(* IEC 61131-3 sources: Everest-Indoor-Unit/SWNOVHIDUOUCR00/SWNOVHIDUOUCR00/Sources/Programs, 17 files *)

(* ---- 020_InputMng.st ---- *)
USING System;
USING System.IO;
USING Libs.IOMng_Basic;
USING Libs.Thermodynamic;
(*
    NOTE:
    In order to ADD a new additional function Analog/Digital Input:
        1. INCREASE THE VALUE OF MAXIMUM NUMBER OF IN/OUT CONSTANT DEFINITON (AIN_NO and DIN_NO)
        2. ADD THE NAME AND UOM IN THE RELATIVE UNION STRUCTURE: AinStruct, AinOffsetStruct and DinStruct.
        3. FROM GLOBAL VARIABLE VIEW FLAG THE NEW PROBE AS PARAMETER AND NFC
*)
VAR_GLOBAL CONSTANT
    (* It's not the number of channels available! *)
    (** Max number of possible Analog Inputs *)
    AIN_NO : USINT := 7;
    (* It's not the number of channels available! *)
    (** Max number of possible Digital Inputs *)
    DIN_NO : USINT := 4;
END_VAR

VAR_GLOBAL
    (**Max n° of Ain used by Local board*)
    MAX_AIN_CH  : USINT;
    (**Max n° of Din used by Local board*)
    MAX_DIN_CH  : USINT;
    (**Max n° of Dout used by Local board*)
    MAX_DOUT_CH : USINT;
    (**Max n° of Aout used by Local board*)
    MAX_AOUT_CH : USINT;
    (**Device parameteres (Number of I/O, type o Core...) *)
    HwDesc_1    : HardwareDescription;

    SystemPressure : REAL;
END_VAR

TYPE
    {REGION DIGITAL INPUT CONFIGURATION}
    DinInfoUnion: UNION
        Fct : DinInfoStruct;
        Arr : ARRAY[1..DIN_NO] OF ErrConfig;
    END_UNION;

    DinInfoStruct: STRUCT
        (**Start/Stop Command*)
        RemOnOff        : ErrConfig;
        (**Flow switch*)
        FlowSw          : ErrConfig;
        (**SG input 1*)
        SG1          : ErrConfig;
        (**SG input 2*)
        SG2          : ErrConfig;
    END_STRUCT;

    DinCfgUnion: UNION
        Fct : DinCfgStruct;
        Arr : ARRAY[1..DIN_NO] OF DinConfig;
    END_UNION;

    DinCfgStruct: STRUCT
        (**Start/Stop Command*)
        RemOnOff        : DinConfig;
        (**Flow switch*)
        FlowSw          : DinConfig;
        (**SG input 1*)
        SG1          : DinConfig;
        (**SG input 2*)
        SG2          : DinConfig;
    END_STRUCT;

    DinData: UNION
        Fct : DinStruct;
        Arr : ARRAY[1..DIN_NO] OF BOOL;
    END_UNION;

    DinStruct: STRUCT
        (**Start/Stop Command*)
        RemOnOff        : BOOL;
        (**Flow switch*)
        FlowSw          : BOOL;
        (**SG input 1*)
        SG1          : BOOL := FALSE;
        (**SG input 2*)
        SG2          : BOOL := FALSE;
    END_STRUCT;
    {ENDREGION}

    {REGION ANALOGIC INPUT CONFIGURATION}
    (*
            PAY ATTENTION!!!
            When you add a new AIN remember to also update the MAIN_UI_SEL and AUX_AIN_TYP enumerators.
        *)

    AinInfoUnion: UNION
        Fct : AinInfoStruct;
        Arr : ARRAY[1..AIN_NO] OF ErrConfig;
    END_UNION;

    AinInfoStruct: STRUCT
        (**BT5 DHW bottom temperature*)
        DHWBottomTemp    :   ErrConfig;
        (**BT4 DHW middle temperature*)
        DHWMiddleTemp    :   ErrConfig;
        (**BT3 DHW top temperature*)
        DHWTopTemp       :   ErrConfig;
        (**BT7 DHW supply temperature*)
        DHWSupplyTemp    :   ErrConfig;
        (**BT1 Outdoor temperature*)
        OutDoorTemp    :   ErrConfig;
        (**BT6 Climate system supply temperature*)
        ClimSupplyTemp    :   ErrConfig;
        (**BP1 System pressure*)
        SysPress    :   ErrConfig;
    END_STRUCT;

    AinCfgUnion: UNION
        Fct : AinCfgStruct;
        Arr : ARRAY[1..AIN_NO] OF AinConfig;
    END_UNION;

    AinCfgStruct: STRUCT
        (**BT5 DHW bottom temperature*)
        DHWBottomTemp     :  AinConfig;
        (**BT4 DHW middle temperature*)
        DHWMiddleTemp    :   AinConfig;
        (**BT3 DHW top temperature*)
        DHWTopTemp       :   AinConfig;
        (**BT7 DHW supply temperature*)
        DHWSupplyTemp    :   AinConfig;
        (**BT1 Outdoor temperature*)
        OutDoorTemp    :   AinConfig;
        (**BT7 Climate system supply temperature*)
        ClimSupplyTemp    :   AinConfig;
        (**BP1 System pressure*)
        SysPress    :   AinConfig;
    END_STRUCT;

    AinData: UNION
        Fct : AinDataStruct;
        Arr : ARRAY[1..AIN_NO] OF REAL;
    END_UNION;

    AinDataStruct: STRUCT
        {ATTRIBUTE UOM CELSIUS}
        {METADATA MAX_VAL 999.9}
        {METADATA MIN_VAL -99.9}
        (**BT5 DHW bottom temperature*)
        DHWBottomTemp       :   REAL;
        {ATTRIBUTE UOM CELSIUS}
        {METADATA MAX_VAL 999.9}
        {METADATA MIN_VAL -99.9}
        (**BT4 DHW middle temperature*)
        DHWMiddleTemp      :   REAL;
        {ATTRIBUTE UOM CELSIUS}
        {METADATA MAX_VAL 999.9}
        {METADATA MIN_VAL -99.9}
        (**BT3 DHW top temperature*)
        DHWTopTemp      :   REAL;
        {ATTRIBUTE UOM CELSIUS}
        {METADATA MAX_VAL 999.9}
        {METADATA MIN_VAL -99.9}
        (**BT7 DHW supply temperature*)
        DHWSupplyTemp      :   REAL;
        {ATTRIBUTE UOM CELSIUS}
        {METADATA MAX_VAL 999.9}
        {METADATA MIN_VAL -99.9}
        (**BT1 Outdoor temperature*)
        OutDoorTemp      :   REAL;
        {ATTRIBUTE UOM CELSIUS}
        {METADATA MAX_VAL 999.9}
        {METADATA MIN_VAL -99.9}
        (**BT6 Climate system supply temperature*)
        ClimSupplyTemp    :   REAL;
        {ATTRIBUTE UOM BAR}
        {METADATA MAX_VAL 7.0}
        {METADATA MIN_VAL -1.0}
        (**BP1 System pressure*)
        SysPress    :   REAL;
    END_STRUCT;

    AinOffset: UNION
        Fct : AinOffSetStruct;
        Arr : ARRAY[1..AIN_NO] OF REAL;
    END_UNION;

    AinOffSetStruct: STRUCT
        {ATTRIBUTE UOM DELTACELSIUS}
        (**BT5 DHW bottom temperature*)
        DHWBottomTemp      :   REAL;
        {ATTRIBUTE UOM DELTACELSIUS}
        (**BT4 DHW middle temperature*)
        DHWMiddleTemp      :   REAL;
        {ATTRIBUTE UOM DELTACELSIUS}
        (**BT3 DHW top temperature*)
        DHWTopTemp         :   REAL;
        {ATTRIBUTE UOM DELTACELSIUS}
        (**BT7 DHW supply temperature*)
        DHWSupplyTemp      :   REAL;
        {ATTRIBUTE UOM DELTACELSIUS}
        (**BT1 Outdoor temperature*)
        OutDoorTemp        :   REAL;
        {ATTRIBUTE UOM DELTACELSIUS}
        (**BT6 Climate system supply temperature*)
        ClimSupplyTemp     :   REAL;
        {ATTRIBUTE UOM BAR}
        (**BP1 System pressure*)
        SysPress           :   REAL;
    END_STRUCT;

    {ENDREGION}
END_TYPE

VAR_GLOBAL PERSISTENT
        ReservedIOCfg :BOOL := TRUE;
        Din_Cfg     : DinCfgUnion  := (Fct := (
            (**StartStop*)
            RemOnOff        := (Ch := 0, ModeType := MODE_TYPE_DIN#LIB_IO_DIN),
            (**Flow switch*)
            FlowSw          := (Ch := 0, ModeType := MODE_TYPE_DIN#LIB_IO_DIN),
            (**SG input 1*)
            SG1          := (Ch := 4, ModeType := MODE_TYPE_DIN#LIB_IO_DIN, logic := TRUE),
            (**SG input 2*)
            SG2          := (Ch := 5, ModeType := MODE_TYPE_DIN#LIB_IO_DIN, logic := TRUE)
        ));

        Ain_Cfg     : AinCfgUnion := (Fct := (
            (**DHW bottom temperature*)
            DHWBottomTemp       := (Ch := 5,  ModeType := MODE_TYPE_AIN#LIB_IO_PROBE_NTC),
            (**DHW middle temperature*)
            DHWMiddleTemp       := (Ch := 4,  ModeType := MODE_TYPE_AIN#LIB_IO_PROBE_NTC),
            (**DHW top temperature*)
            DHWTopTemp          := (Ch := 3,  ModeType := MODE_TYPE_AIN#LIB_IO_PROBE_NTC),
            (**DHW supply temperature*)
            DHWSupplyTemp       := (Ch := 6,  ModeType := MODE_TYPE_AIN#LIB_IO_PROBE_NTC),
            (**Outdoor temperature*)
            OutDoorTemp         := (Ch := 1,  ModeType := MODE_TYPE_AIN#LIB_IO_PROBE_NTC),
            (**Climate system supply temperature*)
            ClimSupplyTemp      := (Ch := 2,  ModeType := MODE_TYPE_AIN#LIB_IO_PROBE_NTC),
            (**System pressure*)
            SysPress            := (Ch := 10,  ModeType := MODE_TYPE_AIN#LIB_IO_PROBE_4_20MA)
        ));

    Ain_Min     : AinData := (Fct := (
        SysPress := 0
    ));

    Ain_Max     : AinData := (Fct := (
        SysPress := 6

    ));

    Ain_Offset  : AinOffset :=();

    (**Probe alarm delay*)
    {ATTRIBUTE UOM SECOND}
    PrbAlrm_DT : UINT(0..999) := 10;
END_VAR

PROGRAM InputMng
    VAR_TEMP
        i : DINT;
    END_VAR

    (*All the Programs are skipped while the default valeus are being installed*)
    IF RestoreDefault THEN
        RETURN;
    END_IF;

    {REGION Analog Input Enable}
        Ain_Cfg.Fct.DHWBottomTemp.Enable := TRUE;
        Ain_Cfg.Fct.DHWMiddleTemp.Enable := TRUE;
        Ain_Cfg.Fct.DHWTopTemp.Enable := TRUE;
        Ain_Cfg.Fct.DHWSupplyTemp.Enable := TRUE;
        Ain_Cfg.Fct.ClimSupplyTemp.Enable := TRUE;
        Ain_Cfg.Fct.OutDoorTemp.Enable := TRUE;
        Ain_Cfg.Fct.SysPress.Enable := TRUE;
    {ENDREGION}

    {REGION Digital Input Enable}
        Din_Cfg.Fct.RemOnOff.Enable := TRUE;
        Din_Cfg.Fct.FlowSw.Enable := TRUE;
        Din_Cfg.Fct.SG1.Enable := TRUE;
        Din_Cfg.Fct.SG2.Enable := TRUE;
    {ENDREGION}

    (*Initialization Probe Alarm Delay*)
    FOR i := LOWER_BOUND(Ain_Cfg.Arr, 1) TO UPPER_BOUND(Ain_Cfg.Arr, 1) DO
        Ain_Cfg.Arr[i].AlrmDT := TO_UDINT(PrbAlrm_DT);
    END_FOR;

    IO_Mng.Read(
        BOARD_TYPE#PCO,
        ID,
        U,
        Din_Cfg.Arr,
        Ain_Cfg.Arr,
        Ain_Max.Arr,
        Ain_Min.Arr,
        Ain_Offset.Arr,
        Din_Data.Arr,
        Din_Info.Arr,
        Ain_Data.Arr,
        Ain_Info.Arr,
        uConfig
    );

    HandleSpecialID(1, LIB_IO_PROBE_U_FREQ, 5, uID1);
    WaterFlow_DHW2 := (TO_REAL(uID1.ui) * 0.0106);    // 530 pulses per litre

    HandleSpecialID(2, LIB_IO_PROBE_U_FREQ, 5, uID2);
    WaterFlow_DHW := (TO_REAL(uID2.ui) * 0.0106);    // 530 pulses per litre

    SystemPressure := To_Real(U[10].ud);
    SystemPressure := To_Real(U[10].ui);
    SystemPressure := To_Real(U[10].b);
    SystemPressure := To_Real(U[10].r);
END_PROGRAM

(* ---- 031_StoreAlarms.st ---- *)
USING System;
USING System.Alarm;
USING System.Timer;
USING System.Math;

USING Libs.Logics;
USING Libs.Alarm_Mng;

TYPE
    (**This structure manages all unit's alarms*)
    AlarmUnion : UNION
        (**Array of FBs Alarm_Req*)
        Arr   : ARRAY [1..noAlrms] OF Alarm_Req;
        (**Table of all alarms and them property*)
        Table : AlarmsStruct;
    END_UNION;

    (**List all alarms and them property (Code, Category, Reset type, ...)*)
    AlarmsStruct : STRUCT
        (**Error in number of permanent memory writes*)
        Al_RetainMemNo : Alarm_Req           	 :=	 (StrCode := 'A01', Info := (Code := 001, Category := CAT_AL_SRS_UNIT, Reset := AlarmResetType#Manual));
        (**DHW bottom temperature*)
        Al_DHWBottomTemp : Alarm_Req             :=  (StrCode := 'A02', Info := (Code := 002, Category := CAT_AL_SRS_UNIT, Reset := AlarmResetType#Auto));
        (**DHW middle temperature*)
        Al_DHWMiddleTemp : Alarm_Req             :=  (StrCode := 'A03', Info := (Code := 003, Category := CAT_AL_SRS_UNIT, Reset := AlarmResetType#Auto));
        (**DHW top temperature*)
        Al_DHWTopTemp : Alarm_Req                :=  (StrCode := 'A04', Info := (Code := 004, Category := CAT_AL_SRS_UNIT, Reset := AlarmResetType#Auto));
        (**DHW supply temperature*)
        Al_DHWSupplyTemp : Alarm_Req             :=  (StrCode := 'A05', Info := (Code := 005, Category := CAT_AL_SRS_UNIT, Reset := AlarmResetType#Auto));
        (**Outdoor temperature*)
        Al_OutDoorTemp    :   Alarm_Req          :=  (StrCode := 'A06', Info := (Code := 006, Category := CAT_AL_SRS_UNIT, Reset := AlarmResetType#Auto));
        (**Climate system supply temperature*)
        Al_ClimSupplyTemp    :   Alarm_Req       :=  (StrCode := 'A07', Info := (Code := 007, Category := CAT_AL_SRS_UNIT, Reset := AlarmResetType#Auto));
        (**System pressure*)
        Al_SysPress    :   Alarm_Req             :=  (StrCode := 'A08', Info := (Code := 008, Category := CAT_AL_SRS_UNIT, Reset := AlarmResetType#Auto));
        (**Outdoor unit offline*)
        Al_OUOffline   : Alarm_Req               :=  (StrCode := 'A09', Info := (Code := 009, Category := CAT_AL_SRS_UNIT, Reset := AlarmResetType#Auto));
        (**FreezeProtectionActive*)
        Al_FreezeProAct   : Alarm_Req            :=  (StrCode := 'A10', Info := (Code := 010, Category := CAT_AL_SRS_UNIT, Reset := AlarmResetType#Auto));
    END_STRUCT;
END_TYPE

VAR_GLOBAL CONSTANT
    {REGION UPDATE EVERY TIME AN ALARM IS ADDEDD!}
        (**Number of alarm saved inside ALARM table.
         *NOTE: update every time an alarm is addedd!
        *)
        noAlrms : UINT := 28;
    {ENDREGION}

    {REGION ALARM LOG CONFIGURATION}
        (**Number of logs of alarms saved inside ALARM-LOG table*)
        noAlrmsLog     : UINT := 20;
        (**
         *Size of the array VARs_TO_LOG.
         *Number of additionals variables saved inside ALARM-LOG table,
         *when an alarm is triggered (NOTE: used inside System.Alarm library)
        *)
        MaxAlarmValues : UINT := 0;
    {ENDREGION}

    {REGION CONFIGURE HERE YOUR ALARMs CATEGORY (max 16). YOU NEED TO USE "ActAlr_ForCategory".}
    (**Alarm category associate to ActAlr_ForCategory BIT_0 *) CAT_AL_SRS_UNIT          : UINT := 1;
    (**Alarm category associate to ActAlr_ForCategory BIT_1 *) CAT_AL_SRS_CIRC1         : UINT := 2;
    (**Alarm category associate to ActAlr_ForCategory BIT_2 *) CAT_WARN_CIRC1           : UINT := 4;
    (**Alarm category associate to ActAlr_ForCategory BIT_3 *) SENSOR                   : UINT := 8;
    (**Alarm category associate to ActAlr_ForCategory BIT_4 *) HEATPUMP                 : UINT := 16;
    (**Alarm category associate to ActAlr_ForCategory BIT_5 *) FREE_0                   : UINT := 32;
    (**Alarm category associate to ActAlr_ForCategory BIT_6 *) FREE_1                   : UINT := 64;
    (**Alarm category associate to ActAlr_ForCategory BIT_7 *) FREE_2                   : UINT := 128;
    (**Alarm category associate to ActAlr_ForCategory BIT_8 *) FREE_3                   : UINT := 256;
    (**Alarm category associate to ActAlr_ForCategory BIT_9 *) FREE_4                   : UINT := 512;
    (**Alarm category associate to ActAlr_ForCategory BIT_10*) FREE_5                   : UINT := 1024;
    (**Alarm category associate to ActAlr_ForCategory BIT_11*) FREE_6                   : UINT := 2048;
    (**Alarm category associate to ActAlr_ForCategory BIT_12*) FREE_7                   : UINT := 4096;
    (**Alarm category associate to ActAlr_ForCategory BIT_13*) FREE_8                   : UINT := 8192;
    (**Alarm category associate to ActAlr_ForCategory BIT_14*) FREE_9                   : UINT := 16384;
    (**Alarm category associate to ActAlr_ForCategory BIT_15*) FREE_10                  : UINT := 32768;
    {ENDREGION}
END_VAR

VAR_GLOBAL PERSISTENT
    (**Log alarm array*)
    Log_Alarm  : ARRAY[1..noAlrmsLog] OF AlarmLog;
    (**Index of Log_Alarm *)
    LogAlrmIdx : UINT;
END_VAR

VAR_GLOBAL
    {REGION ALARMS MANAGEMENT}
        (**Container of Alarms table*)
        Alarms              : AlarmUnion;
        (**Array of active alarms*)
        Active_Alrm         : ARRAY[1..noAlrms] OF UINT;
        (**Active alarm status for each category, max 16 differents category (Bit15..Bit0)*)
        ActAlr_ForCategory  : WORD;
    {ENDREGION}

    {REGION ALARMS LOG}
        (**Array of variables to store inside LOG_ALARM array, when an alarm happen*)
        VARs_TO_LOG : ARRAY[0..MaxAlarmValues] OF AlarmValue;
        (**Empty structured used to clean LOG_ALARM array*)
        CleanLog    : AlarmLog;
    {ENDREGION}
END_VAR

VAR_GLOBAL INTERNAL
    (*Used by Modbus files transfer protocol*)
    AlrmInfoArr : ARRAY [1..noAlrms] OF AlarmInfo;
END_VAR

(**This program manages alarm categories and detects the alarms*)
PROGRAM StoreAlarms
    VAR_TEMP
        (**Numeber of alarm active*)
        TotActAlm : UINT;
    END_VAR

    VAR
        (**Array index*)
        idx             : DINT;
        (**Numeber of alarm active in previous cycle*)
        TotActAlm_Old   : UINT;
        TP_ResAlrmByBMS : TP;

        {REGION USED BY LOG-ALARM TO STORE THE "ADDITIONAL VARIABLES"}
        (**A42 trigger used to store additional values*)
        RFtrg_Alr1          : RF_TRIG;
        (**A48 trigger used to store additional values*)
        RFtrg_Alr2          : RF_TRIG;
        (**A46 trigger used to store additional values*)
        RFtrg_Alr3          : RF_TRIG;
        (**A43 trigger used to store additional values*)
        RFtrg_Alr4          : RF_TRIG;
        (**A01 trigger used to store additional values*)
        RFtrg_Alr5          : RF_TRIG;
        (**A35 trigger used to store additional values*)
        RFtrg_Alr6          : RF_TRIG;
        (**A32 trigger used to store additional values*)
        RFtrg_Alr7          : RF_TRIG;
        (**A33 trigger used to store additional values*)
        RFtrg_Alr8          : RF_TRIG;
        (**A37 trigger used to store additional values*)
        RFtrg_Alr9          : RF_TRIG;
        (**A34 trigger used to store additional values*)
        RFtrg_Alr10         : RF_TRIG;
        {ENDREGION}
    END_VAR

    (*Alarm management is be skipped while the default valeus are being installed OR at startup while I/O are being read*)
    IF RestoreDefault OR UnitStatus = UNIT_STATUS#Wait THEN
        RETURN;
    END_IF;

    {REGION RESET ALARM ARRAY}
    TP_ResAlrmByBMS(IN := ResAlrmByBMS, PT := T#5s);        (*Request of reset by BMS*)
    ResAlrmByBMS := TP_ResAlrmByBMS.Q;

    AlrmRes := ResAlrmByBMS OR ResAlrmByHMI;
    {ENDREGION}

    {REGION CLEAN THE LOG ARRAY}
    IF LogAlrmRes THEN
        LogAlrmRes       := FALSE;
        (*RESTART LOG*)
        LogAlrmIdx := 0;

        (*CLEAR LOG LIST*)
        FOR idx := 1 TO TO_DINT(UPPER_BOUND(Log_Alarm, 1)) DO
            Log_Alarm[idx] := CleanLog;
        END_FOR;
    END_IF;
    {ENDREGION}

    {REGION SET DYNAMIQUE CATEGORY}

    {ENDREGION}

    {REGION GET ACTIVE ALARMS}
    FOR idx := 1 TO UPPER_BOUND(Alarms.Arr, 1) DO
        (*Copy the alarm info into a dedicated array*)
        AlrmInfoArr[idx] := Alarms.Arr[idx].Info;

        {REGION "ADDITIONAL VARIABLES" stored inside LOG_ALARM array, when an alarm happen}
		/*IF Alarms.Arr[idx].Info.Code = Alarms.Table.Al_Envelope_Circ1.Info.Code THEN
			RFtrg_Alr1(CLK := Alarms.Arr[idx].Info.Trigger);
            IF RFtrg_Alr1.Q THEN
                VARs_TO_LOG[0].UINT := TO_UINT(0);
            END_IF;*/
		/*ELSIF Alarms.Arr[idx].Info.Code = Alarms.Table.Al_Inv_Circ1.Info.Code THEN
			RFtrg_Alr2(CLK := Alarms.Arr[idx].Info.Trigger);
            IF RFtrg_Alr2.Q THEN
                    VARs_TO_LOG[0].UINT := PWRP_ErrCode_Circ1;
            END_IF;*/
		/*ELSIF Alarms.Arr[idx].Info.Code = Alarms.Table.Al_HiDscgTempComp1_Circ1.Info.Code THEN
        	RFtrg_Alr3(CLK := Alarms.Arr[idx].Info.Trigger);
            IF RFtrg_Alr3.Q THEN
                VARs_TO_LOG[0].UINT := TO_UINT(DscgT_Zone_Circ1);
            END_IF;*/
		/*ELSIF Alarms.Arr[idx].Info.Code = Alarms.Table.Al_DisStartDp_Circ1.Info.Code THEN
			RFtrg_Alr4(CLK := Alarms.Arr[idx].Info.Trigger);
            IF RFtrg_Alr4.Q THEN
                VARs_TO_LOG[0].REAL := DeltaP_Circ1;
            END_IF;*/
		/*ELSIF Alarms.Arr[idx].Info.Code = Alarms.Table.Al_RetainMemNo.Info.Code THEN
			RFtrg_Alr5(CLK := Alarms.Arr[idx].Info.Trigger);
            IF RFtrg_Alr5.Q THEN
                VARs_TO_LOG[0].UDINT := TO_UDINT(RetainMemWrites);
            END_IF;*/
		/*ELSIF Alarms.Arr[idx].Info.Code = Alarms.Table.Al_EEV_Circ1.Info.Code THEN
			RFtrg_Alr6(CLK := Alarms.Arr[idx].Info.Trigger);
            IF RFtrg_Alr6.Q THEN
                VARs_TO_LOG[0].UINT := TO_UINT(EEV_AlrmCode_Circ1);
            END_IF;*/
		/*ELSIF Alarms.Arr[idx].Info.Code = Alarms.Table.Al_WkrHrsComp1_Circ1.Info.Code THEN
			RFtrg_Alr7(CLK := Alarms.Arr[idx].Info.Trigger);
            IF RFtrg_Alr7.Q THEN
                VARs_TO_LOG[0].UINT := TO_UINT(Comp1Circ1_HrsRetain);
            END_IF;*/
		/*ELSIF Alarms.Arr[idx].Info.Code = Alarms.Table.Al_WkrHrsSrc_Circ1.Info.Code THEN
			RFtrg_Alr10(CLK := Alarms.Arr[idx].Info.Trigger);
            IF RFtrg_Alr10.Q THEN
                VARs_TO_LOG[0].UINT := TO_UINT(Source1Circ1_HrsRetain);
            END_IF;*/
		//END_IF;
        {ENDREGION}

        Alarms.Arr[idx]
                        (
                            DataVal         := VARs_TO_LOG, (* Remember to define ALARM_VALUES *)
                            AlrmRes         := AlrmRes,
                            Lst_ActAlrm     := Active_Alrm,
                            Lst_LogAlrm     := Log_Alarm,
                            Lst_LogAlrm_Idx := LogAlrmIdx
                        );
    END_FOR;
    {ENDREGION}

    {REGION GET ALARM CATEGORIES}
    ActAlr_ForCategory := Alarm_Mng(Active_Alrm);
    Al_SrsUnit            := ActAlr_ForCategory.0;  									// BIT n.0  -> CAT_AL_SRS_UNIT
    Al_SrsCirc1           := ActAlr_ForCategory.1 OR Al_SrsUnit;// BIT n.1  -> Al_SRS_CIRC1
    Wrg_Regul             := ActAlr_ForCategory.4;                      				// BIT n.4  -> CAT_WRG_REGUL
    Wrg_Circ1             := ActAlr_ForCategory.5;                      				// BIT n.7  -> CAT_WRG_CIRC1
    Wrg_HrsCounters       := ActAlr_ForCategory.7;                      				// BIT n.10 -> CAT_WRG_HRSCOUNTER
    {ENDREGION}

    {REGION MANAGEMENT OF ALARM RELAY AND GROUPED ALARMS}
    (*Depending on alarm relay configuration, the alarm relay is activated by serious alarms only or by all alarms (including devices maintenance, retain memory,...) *)
    Al_RegulationAlrms :=    Al_SrsUnit
                          OR Al_SrsCirc1
                          OR Wrg_Regul;

    Al_MiscAlrms :=    Wrg_Circ1
                    OR Wrg_HrsCounters;

    RelayAlrm := Al_RegulationAlrms OR Al_MiscAlrms;
    {ENDREGION}

    {REGION COUNT OF TOTAL ALARMs AND WARNINGs ACTIVE}
    FOR idx := 1 TO TO_DINT(UPPER_BOUND(Active_Alrm,1)) DO
        IF Active_Alrm[idx] >= 1 THEN
            TotActAlm := TotActAlm + 1;
        END_IF;
    END_FOR;

    GblAlarm := UINT_TO_BOOL(TotActAlm);

    (*LED-ALARM and BUZZER*)
    IF TotActAlm > TotActAlm_Old THEN
        Req_FixLED_Alarm   := FALSE;    // LED-ALARM on
        Req_BlinkLED_Alarm := TRUE;     // LED-ALARM is blinking
        BuzzerSilenced     := FALSE;    // Buzzer is buzzing
    END_IF;

    TotActAlm_Old := TotActAlm;
    {ENDREGION}
END_PROGRAM

(* ---- 120_OutputMng.st ---- *)
USING System.IO;
USING System;
USING Libs.Math;
USING Libs.IOMng_Basic;

(*
    NOTE:
    In order to ADD a new additional function Analog/Digital Output:
        1. INCREASE THE VALUE OF MAXIMUM NUMBER OF IN/OUT CONSTANT DEFINITON (MAX_DO_NO and MAX_AO_NO)
        2. ADD THE NAME AND UOM IN THE RELATIVE UNION STRUCTURE: AoutStruct and DoutStruct
        3. FROM GLOBAL VARIABLE VIEW FLAG THE NEW PROBE AS PARAMETER AND NFC
*)
VAR_GLOBAL CONSTANT
    (* It's not the number of channels available! *)
    (** Max number of possible Digital Outputs *)
    MAX_DO_NO   : USINT := 7;
    (* It's not the number of channels available! *)
    (** Max number of possible Analog Outputs *)
    MAX_AO_NO   : USINT := 2;
END_VAR

TYPE
    {REGION ANALOGIC OUTPUT CONFIGURATION}
        AoutInfoUnion: UNION
            Fct : AoutInfoStruct;
            Arr : ARRAY[1..MAX_AO_NO] OF ErrConfig;
        END_UNION;

        AoutInfoStruct: STRUCT
            (**Circulation pump 1*)
            CircPump1    :   ErrConfig;
            (**Circulation pump 2*)
            CircPump2    :   ErrConfig;
        END_STRUCT;

        AoutCfgUnion: UNION
            Fct : AoutCfgStruct;
            Arr : ARRAY[1..MAX_AO_NO] OF AoutConfig;
        END_UNION;

        AoutCfgStruct: STRUCT
            (**Circulation pump 1*)
            CircPump1    :   AoutConfig;
            (**Circulation pump 2*)
            CircPump2    :   AoutConfig;
        END_STRUCT;

        AoutData: UNION
            Fct : AoutStruct;
            Arr : ARRAY[1..MAX_AO_NO] OF REAL;
        END_UNION;

        AoutStruct: STRUCT
            (**Circulation pump 1*)
            {ATTRIBUTE UOM PERCENT}
            CircPump1    :   REAL;
            {ATTRIBUTE UOM PERCENT}
            (**Circulation pump 2*)
            CircPump2    :   REAL;
        END_STRUCT;
    {ENDREGION}

    {REGION DIGITAL OUTPUT CONFIGURATION}
        DoutInfoUnion: UNION
            Fct : DoutInfoStruct;
            Arr : ARRAY [1..MAX_DO_NO] OF ErrConfig;
        END_UNION;

        DoutInfoStruct: STRUCT
            (**General alarm *)
            GlbAl          :   ErrConfig;
            (**Shunt valve*)
            ShuntVlvDout          :   ErrConfig;
            (**Immersion heater step 1*)
            ImmheatStep1   : ErrConfig;
            (**Immersion heater step 2*)
            ImmheatStep2   : ErrConfig;
            (**Immersion heater step 3*)
            ShuntVlvOffDout   : ErrConfig;
            (**Reversing valve*)
            RevVlv         : ErrConfig;
            (**Shut off valve*)
            ShutOffVlv     : ErrConfig;
        END_STRUCT;

        DoutCfgUnion: UNION
            Fct : DoutCfgStruct;
            Arr : ARRAY [1..MAX_DO_NO] OF DoutConfig;
        END_UNION;

        DoutCfgStruct: STRUCT
            (**General alarm *)
            GlbAl          :    DoutConfig;
            (**Shunt valve*)
            ShuntVlvDout          :   DoutConfig;
            (**Immersion heater step 1*)
            ImmheatStep1   : DoutConfig;
            (**Immersion heater step 2*)
            ImmheatStep2   : DoutConfig;
            (**Immersion heater step 3*)
            ShuntVlvOffDout   : DoutConfig;
            (**Reversing valve*)
            RevVlv         : DoutConfig;
            (**Shut off valve*)
            ShutOffVlv     : DoutConfig;
        END_STRUCT;

        DoutData: UNION
            Fct : DoutStruct;
            Arr : ARRAY[1..MAX_DO_NO] OF BOOL;
        END_UNION;

        DoutStruct: STRUCT
            (**General alarm *)
            GlbAl               :   BOOL;
            (**Shunt valve*)
            ShuntVlvDout            :   BOOL;
            (**Immersion heater step 1*)
            ImmheatStep1   : BOOL;
            (**Immersion heater step 2*)
            ImmheatStep2   : BOOL;
            (**Immersion heater step 3*)
            ShuntVlvOffDout   : BOOL;
            (**Reversing valve*)
            RevVlv         : BOOL;
            (**Shut off valve*)
            ShutOffVlv     : BOOL;
        END_STRUCT;
    {ENDREGION}

END_TYPE

VAR_GLOBAL PERSISTENT
    Dout_Cfg        : DoutCfgUnion  := (Fct := (
        (**General alarm *)
        GlbAl               := (Ch := 0),
        (**Shunt valve*)
        ShuntVlvDout        := (Ch := 8),
        (**Immersion heater step 1*)
        ImmheatStep1        := (Ch := 4),
        (**Immersion heater step 2*)
        ImmheatStep2        := (Ch := 5),
        (**Immersion heater step 3*)
        ShuntVlvOffDout     := (Ch := 9),
        (**Reversing valve*)
        RevVlv              := (Ch := 1),
        (**Shut off valve*)
        ShutOffVlv          := (Ch := 7)
    ));

    Aout_Cfg        : AoutCfgUnion := (Fct := (
        (**Circulation pump 1*)
        CircPump1      := (Ch := 3,  ModeType := MODE_TYPE_AOUT#LIB_IO_PWM_2_KHZ),
        (**Circulation pump 2*)
        CircPump2      := (Ch := 4,  ModeType := MODE_TYPE_AOUT#LIB_IO_PWM_2_KHZ)

    ));

    Aout_Min : AoutData :=(Fct := (CircPump1 :=0, CircPump2 := 0));
    Aout_Max : AoutData :=(Fct := (CircPump1 :=100, CircPump2 := 100));
END_VAR

PROGRAM OutputMng
    VAR_TEMP
        i : DINT;
    END_VAR
    (*Enabling Analog outputs*)
    {REGION Analog Output Enable}
        Aout_Cfg.Fct.CircPump1.Enable := TRUE;
        Aout_Cfg.Fct.CircPump2.Enable := TRUE;
    {ENDREGION}

    (*Enabling Digital outputs*)
    {REGION Digital Output Enable}
        Dout_Cfg.Fct.GlbAl.Enable := TRUE;
        Dout_Cfg.Fct.ShuntVlvDout.Enable := TRUE;
        Dout_Cfg.Fct.ImmheatStep1.Enable := ImmHeatStage >= 1;
        Dout_Cfg.Fct.ImmheatStep2.Enable := ImmHeatStage >= 2;
        Dout_Cfg.Fct.ShuntVlvOffDout.Enable := TRUE;
        Dout_Cfg.Fct.RevVlv.Enable := TRUE;
        Dout_Cfg.Fct.ShutOffVlv.Enable  := TRUE;
    {ENDREGION}

	{REGION Analog Output value}
    Aout_Data.Fct.CircPump1 := Circ1Act_Req;
    Aout_Data.Fct.CircPump2 := Circ2Act_Req;
	{ENDREGION}

	{REGION Digital Output Value}
	Dout_Data.Fct.GlbAl := GblAlarm;
    Dout_Data.Fct.ShuntVlvDout := ShuntVlv_On;
    Dout_Data.Fct.ImmheatStep1 := ActImmStep_Out.0;
    Dout_Data.Fct.ImmheatStep2 := ActImmStep_Out.1;
    Dout_Data.Fct.ShuntVlvOffDout := ShuntVlv_Off;
    Dout_Data.Fct.RevVlv       := (DHWReq AND OU_CompOn) OR SWValveManA;
    Dout_Data.Fct.ShutOffVlv   := CoolReq OR ShutOffMan;
	{ENDREGION}
    FOR i := 1 TO UPPER_BOUND(Aout_Data.Arr, 1) DO
        Aout_Data.Arr[i] := ScalerLimited(Aout_Data.Arr[i], 0.0, 100.0, Aout_Min.Arr[i], Aout_Max.Arr[i]);
    END_FOR;

    IO_Mng.Write(
        BOARD_TYPE#PCO,
        Dout_Cfg.Arr,
        Dout_Data.Arr,
        Aout_Cfg.Arr,
        Aout_Data.Arr,
        Dout_Info.Arr,
        Aout_Info.Arr,
        NO,
        noConfig,
        Y,
        yConfig,
        uConfig,
        Uout
    );

END_PROGRAM

(* ---- 010_GENERAL_MNG.st ---- *)
USING System;
USING System.NVRAM;
USING System.Timer;
USING System.Serial;
USING System.Globalization;
USING Libs.GetTime;

PROGRAM Main
    VAR
        (**After restoring the memory to default, it waits 6s before restarting the PLC*)
        TON_WaitRestartPlc  : TON;
        (**R_TRIG Restore Default Settings*)
        Rtrg_RestoreDefault  : R_TRIG;
        (**First cycle done used by NVRAM management*)
        FirstCycleDone_NVRAM : BOOL;
        (**Istance of SoftwareSafeUpload manage the system call GetFullDownloadRequest()*)
        SwSafeUpload         : SoftwareSafeUpload;
        i                    : DINT;
    END_VAR

    VAR_TEMP
        NVRAM_BOOL_Tmp : BYTE;
        TmpTimezone : STRING;
    END_VAR

    RetainMemWrites := GetRetainWritingsNumber();

    TaskMainCurrT   := GetTaskStartTimeAdv();
    TaskMainLiveCnt := GetTaskLiveCounter();
    RetainWrN       := TO_UDINT(GetRetainWritingsNumber());
    TaskMainExeT    := TaskMainCurrT - MemTime;
    MemTime         := TaskMainCurrT;

    {REGION RESTORE MEMORY}
    Rtrg_RestoreDefault(CLK := RestoreDefault);
    (*Saving BMS before restoring memory*)
    IF Rtrg_RestoreDefault.Q THEN
        SPV_Addr_SavedRAM := SPV_Addr;
        SPV_Baud_SavedRAM := SPV_Baud;
        SPV_Conf_SavedRAM := SPV_Conf;
    END_IF;

    IF RestoreDefault AND NOT RetainRestored THEN
        RetainRestoreDefault(); (*NOTE: This request will be executed at END of MAIN task.*)
        RetainRestored := TRUE;
    END_IF;

    //------------------------------------------------------------------------------------
    //------------ WARM SOFTWARE RESET----------------------------------------------------
    //------------------------------------------------------------------------------------
    TON_WaitRestartPlc(IN := RetainRestored, PT := T#6s);

    IF TON_WaitRestartPlc.Q THEN
        // Wait 6s because Retain will be write every 5s
        // 0 - WARM start;
        SoftwareReset(0);
    END_IF;
    {ENDREGION}

    {REGION DATE AND TIME}
    GetLocalTime(LocTime);
    Day_Week := DAY_OF_WEEK(LocTime);

    {REGION SET CLOCK TIME BY APPLICA}
    IF AppSetDateTime THEN
        AppSetDateTime := FALSE; //CS: da provare senza il reset
        //Necessary and in this order
        SetTimeZone(AppTimeZone);
        SetTime(AppDateTime); //APPLICA give UTC Times
        TimezoneIdx := FindTimezoneIndex(TimeZonePOSIX, AppTimeZone);
    END_IF;
    {ENDREGION}

    {REGION SET CLOCK TIME BY USER INTERFACE}
    IF SetClock THEN
        SetClock := FALSE;
        //Necessary and in this order
        SetTimeZone(TimeZonePOSIX[TimezoneIdx]);
        SetLocalTime(CONCAT_DT(
		    TO_UINT(YearIn) + 2000,
		    TO_UINT(MonthIn),
		    TO_UINT(DayIn),
		    TO_UINT(HourIn),
		    TO_UINT(MinuteIn),
		    TO_UINT(SecondIn),
		    0
		));
    END_IF;
    {ENDREGION}
    {ENDREGION}

    {REGION RETAIN WRITING SETTINGS}
    (*This FB manage the "retain writing error" as bios specification. *)
    RetainSetErasureWindowSize(ErasureWindowSize);
    RetainSetErasureWindowsNumber(ErasureWindowsNumber);
    RetainSetMaxErasure(MaxErasure);
    {ENDREGION}

    {REGION SYSTEM INFORMATION}
    IF NOT FirstCycleDone THEN
        MemTime        := TaskMainCurrT;
        GetSystemInfo(SysInfo);
        GetHardwareDescription(HardwareInfo);
        GetModel(DeviceType, BoardType, MachineType, HwCode);
        GetProjectInfo(InfoProject);
        GetProductInfo(InfoProduct);
        GUID := SplitPrjGUID(InfoProject.ProjectID);
        SwVersion := (TO_UINT(InfoProject.VersionMajor) * 10000) + (TO_UINT(InfoProject.VersionMinor) * 1000) + TO_UINT(InfoProject.VersionBuild);
		OS_Version := TO_UINT(SysInfo.FirmwareVersion);
		BootVersion := TO_UINT(SysInfo.BootloaderVersion);

        {REGION COMUNICATION IS STOPPED DURING INITIALIZATION OF INTERNAL PROTOCOLs STRUCTUREs.}
        (*BMS*)
        Supervisor.Init(FALSE);
        (*Fieldbus*)
        MBM_Line.Init(FALSE);
        (*Display*)
        Display.Init();
        {ENDREGION}

        {REGION IoT Third Parts Integration: Alarms retrieved via "Modbus File Transfer"}
        (*Following APIs calls are needed*)
        System.Alarm.AlarmInfoManagement(AlrmInfoArr);
        System.Alarm.AlarmLogManagement(LOG_ALARM);
        {ENDREGION}

        {REGION SAVING OF TIMEZONE WHEN RTC SET BY APPs}
		GetTimeZone(TmpTimezone);
        TimezoneIdx := FindTimezoneIndex(TimeZonePOSIX, TmpTimezone);
        {ENDREGION}
        FirstCycleDone := TRUE;
    END_IF;
    {ENDREGION}

    {REGION SYSTEM CONFIGURAITON}
        //System configuration selection
        //None selected
        // 1: Heating system 1 + DHW
        // 2: Heating system 1 + DHW
        // 3: Heating system 1 + Heating system 2 + DHW
        // 4: Heating system 1 + Cooling + DHW
        // 5: Heating system 1 + Heating system 2 + DHW + Cooling

        IF(SystemCfg > 0)THEN
            SystemCfg_AllowDHW := SystemCfg >= 1;
            SystemCfg_AllowHeat := SystemCfg >= 2;
            SystemCfg_AllowImm := SystemCfg >= 1;
            SystemCfg_AllowCool := SystemCfg >=  4;
            SystemCfg_NoCfgSel := FALSE;
        ELSE
            SystemCfg_AllowDHW := FALSE;
            SystemCfg_AllowHeat := FALSE;
            SystemCfg_AllowImm := FALSE;
            SystemCfg_AllowCool := FALSE;
            SystemCfg_NoCfgSel := TRUE;
        END_IF;
    {ENDREGION}

    {REGION PROTOCOLS}

    {REGION BMS/FIELDBUS SERIAL PORTs CONFIGURATION}
    CASE UoMZoneHMI OF
        UOM_ZONE#SI:
            Supervisor.Info.Zone := SI;
            // Server BMS uses only SI to communicate (Client FielBus <-> Server BMS)
            // NOTE: In a net CLIENT+SERVER set NoConverion =0 beetwen: Client FielBus <-> Server BMS to increase pCO speed
            // i.e.: FBnet.Info.Zone=0 and BMSnet.Info.Zone=0
            Display.Info.Zone := SI;
        UOM_ZONE#Imperial:
            Supervisor.Info.Zone := Imperial;
            Display.Info.Zone := Imperial;
    ELSE
        Supervisor.Info.Zone := NONE;
        Display.Info.Zone := NONE;
    END_CASE;

    {REGION CHANGE BMS2 SETTINGS}
    (*Memory after deleting command is immediately ready the next cycles*)
    IF RetainRestored THEN
        // Restore BMS2 settings
        SPV_Addr := SPV_Addr_SavedRAM;
        SPV_Baud := SPV_Baud_SavedRAM;
        SPV_Conf := SPV_Conf_SavedRAM;

        // Force update BMS2 settings
        SPV_ChangeSet := TRUE;
    END_IF;

    IF SPV_ChangeSet THEN
		Supervisor.Info.TimeOut := TO_UDINT(SPV_OfflineTimeout)*1000;
        SetupSerialSettings(Supervisor.SerialSettings, SPV_Baud, SPV_Conf, getServerPort(SPV_Port));
        Supervisor.ChangeIdent(SPV_Addr);
        // Change setting of BMS supervisor port
        Supervisor.ChangeSettings();
        // Set the same settings for BMS port on Default app (NOTE: In case of FW ugrade the device will be reachable with the previous settings)
        SaveIdePortSettings(Supervisor.SerialSettings.Channel, Supervisor.SerialSettings.Speed, Supervisor.SerialSettings.Bits, Supervisor.SerialSettings.Parity, Supervisor.SerialSettings.Stops, SPV_Addr);

        SPV_ChangeSet := FALSE;
    END_IF;

    SPV_Online := Supervisor.Info.Online;
    {ENDREGION}

    {REGION CHANGE FIELDBUS2 SETTINGS}
    IF FB2_ChangeSet THEN
        SetupSerialSettings(MBM_Line.SerialSettings, FB2_Baud, FB2_Conf, getClientPort(MBM_Line_Port));
        // Change setting of FB supervisor port
        MBM_Line.ChangeSettings();

        FB2_ChangeSet := FALSE;
    END_IF;
    {ENDREGION}
    {ENDREGION}

    {REGION READ BUFFER OF EACH SERIAL PORT}
    // NOTE: when the protocols are in START the read() method obtain the variables
    //       from each buffer -> so the variables can be used inside STone.

    // BMS
    Supervisor.Read();
    // Fieldbus
    MBM_Line.Read();
    Display.Read();
	{IF DEF (PGD)}
    	TerminalDetector.Run(Display);
	{ENDIF}
    {ENDREGION}
	{ENDREGION}

    {REGION NVRAM management}
    IF NOT FirstCycleDone_NVRAM THEN

        /*NVRAM_ReadVar(1, NVRAM_BOOL_Tmp);
        Dout_FourWVlv_NVRAM := TO_BOOL(NVRAM_BOOL_Tmp);

        FirstCycleDone_NVRAM := TRUE;
    ELSE
        NVRAM_WriteVar(1, TO_BYTE(Dout_FourWVlv_NVRAM));*/
    END_IF;
    {ENDREGION}

    //Outdoor unit status management
    OU_Online := OU_Unit.Info.isOnline;

    (*Call of SoftwareSafeUpload manage the system call GetFullDownloadRequest()*)
    SwSafeUpload(
        KeybOffOn := BmsOnOff,
        StartUpload := UnitOff
    );
END_PROGRAM

(* ---- 030_AlarmsMng.st ---- *)
USING System;
USING System.Timer;
USING Libs.Timer;

PROGRAM AlarmsMng
	VAR
	    RTrig_RetainErr : R_TRIG;
	END_VAR

    (*Alarm management is skipped while the default valeus are being installed OR at startup while I/O are being read*)
    IF RestoreDefault OR UnitStatus = UNIT_STATUS#Wait THEN
        RETURN;
    END_IF;

	RTrig_RetainErr(
		CLK := ExceptionInstance.ExceptionError = ERR_RETAIN_SAVE_TOO_OFTEN
	);
	Alarms.Table.Al_RetainMemNo.Info.Trigger := RTrig_RetainErr.Q;

    {REGION UNIT ALARMS BY DIN}
    {ENDREGION}

    {REGION PROBES ALARMS}
    Alarms.Table.Al_DHWBottomTemp.Info.Trigger := Ain_Info.Fct.DHWBottomTemp.Trigger;
    Alarms.Table.Al_DHWMiddleTemp.Info.Trigger := Ain_Info.Fct.DHWMiddleTemp.Trigger;
    Alarms.Table.Al_DHWTopTemp.Info.Trigger := Ain_Info.Fct.DHWTopTemp.Trigger;
    Alarms.Table.Al_DHWSupplyTemp.Info.Trigger := Ain_Info.Fct.DHWSupplyTemp.Trigger;
    Alarms.Table.Al_ClimSupplyTemp.Info.Trigger := Ain_Info.Fct.ClimSupplyTemp.Trigger;
    Alarms.Table.Al_OutDoorTemp.Info.Trigger := Ain_Info.Fct.OutDoorTemp.Trigger;
    Alarms.Table.Al_SysPress.Info.Trigger := Ain_Info.Fct.SysPress.Trigger;
    Alarms.Table.Al_OUOffline.Info.Trigger := OU_ComError;
    {ENDREGION}

    {REGION OUTDOOR UNIT ALARMS}
    IF NOT NoOutdoorUnit THEN

    END_IF;

    {ENDREGION}

    {REGION LOGIC ALARMS}
    Alarms.Table.Al_FreezeProAct.Info.Trigger := CS_FreezeProtAct;
    {ENDREGION}

END_PROGRAM

(* ---- 040_OnOffUnit.st ---- *)
USING System.Timer;
USING Libs.Thermodynamic;

PROGRAM OnOffUnit
    VAR
        (**Instance TON to manage startup delay for I/O*)
        TON_StartUpDT : TON;
    END_VAR

    (*All the Programs are skipped while the default valeus are being installed*)
    IF RestoreDefault THEN
        RETURN;
    END_IF;

    (*This delay is used to give the time to other parts of the application to initialize (e.g. I/O to be configured)*)
    TON_StartUpDT(
        IN := TRUE,
        PT := T#5s
    );

    (*UNIT ON/OFF COMMAND*)
    UnitOn := TRUE;
//                AND NOT Al_SrsUnit
//                AND (BmsOnOff OR NOT En_SPV_OnOff)
//                AND (Din_Data.Fct.RemOnOff OR NOT Din_Info.fct.RemOnOff.configured);

    UnitOff := NOT UnitOn;
    IF UnitOff THEN
        UnitOn := TRUE;
        /*EEV_Circ1_Man_En := FALSE;
        Comp1_Circ1_ManModeEn := FALSE;
        Src_En_Man := FALSE;*/
    END_IF;

    //ManMode := EEV_Circ1_Man_En OR Comp1_Circ1_ManModeEn OR Src_En_Man;

    {REGION UNIT STATUS}
    IF NOT(TON_StartUpDT.Q) THEN
        (*Wait*)
        UnitStatus          := UNIT_STATUS#Wait;
    ELSIF Al_SrsUnit THEN
        (*Off By Alarm*)
        UnitStatus          := UNIT_STATUS#OffByAlarm;
    ELSIF NOT(BmsOnOff) AND En_SPV_OnOff THEN
        (*Off By BMS*)
        UnitStatus          := UNIT_STATUS#OffByBMS;
    ELSIF (NOT(Din_Data.Fct.RemOnOff) AND Din_Info.Fct.RemOnOff.configured) THEN
        (*Off By Digital Input*)
        UnitStatus          := UNIT_STATUS#OffByDI;
    ELSIF NOT(KeybOnOff) THEN
        (*Off By Keyboard*)
        UnitStatus          := UNIT_STATUS#OffByKeyboard;
    ELSIF ManMode THEN
        (*Unit manual mode active*)
        UnitStatus          := UNIT_STATUS#Manual;
    ELSIF UnitOn THEN
        (*Unit ON*)
        UnitStatus          := UNIT_STATUS#UnitON;
    END_IF;
    {ENDREGION}

END_PROGRAM

(* ---- 050_RegulationMode.st ---- *)
USING System;
USING System.Math;
USING Libs.Math;
USING Libs.PID_Incr;
USING Libs.Timer;

VAR_GLOBAL
        (**DHW switch due to timer*)
        DHWFrcSwitch            : BOOL;
          (**DHW transition timer*)
        TON_DHWTimer            : TON_s;
        (**Allow/block OU from energybalance*)
        SR_Energybalance_HP        : SR;
        (**Allow/block OU from energybalance*)
        SR_Energybalance_CH        : SR;
        (**Switch to cooling*)
        SwToCoolReq                : BOOL;
END_VAR

PROGRAM RegulationMode
    VAR
        (**Iteration value*)
        i                       : INT;
        (**Iteration value*)
        j                       : INT;
        (**Iteration value*)
        k                       : INT;
        (**Outside temperature sample timer*)
        TON_OutDoorTemp         : TON_S;
        (**First full FilterHrs temperature samples taken*)
        OutDoorTempAvgReady     : BOOL;

        OutDoorTempFilterTmp    : REAL;
        (**Outside temperature Sensor sample timer*)
        TON_OutDoorTempSnsr     : TON_S;
        (**Comp minimum running time in heat or cool mode*)
        TON_MinRunTime          : TON_s;
        MinRunTime              : BOOL;
        (**DHW switch complete*)
        DHWFrcSwitchDone        : BOOL;
        (**Disable regular state transition during DHW switch*)
        Dis_OpStateSwitch       : BOOL;
        (**RS latch Comp minimum running time in heat or cool mode*)
        RS_ChangeOfMode         : RS;
        (**SG status byte*)
        SG_Status_Byte          : BYTE;
        (**Energy balance timer*)
        TON_Energybalance       : TON_S;
        (**Disable automode*)
        Dis_AutoMode            : BOOL;
        (**FirstCycle*)
        FirstCycle              : BOOL := 1;
        (**Outdoor sensor average collected*)
        OutDoorTempSnsrAvgReady : BOOL;

        OutDoorTempSnsr_FiltSec : INT := 100;
        (**Outdoor temporary starage af collected values*)
        OutDoorTempSnsrFilter_PreCalc : ARRAY [0..300] OF REAL;

    END_VAR

    //Jump logic during startup to avoid incorrect I/O value sampling
    IF RestoreDefault OR UnitStatus = UNIT_STATUS#Wait THEN
        RETURN;
    END_IF;

    {REGION SMARTGRID INPUT MANAGEMENT}
        SG_Status_Byte.0 := Din_Data.Fct.SG1 AND SGActive;
        SG_Status_Byte.1 := Din_Data.Fct.SG2 AND SGActive;
        SG_Status := TO_USINT(SG_Status_Byte);
    {ENDREGION}

    {REGION OUTDOOR TEMPERATURE FILTER CALCULATION}

        //Update temperature value every 5 minute or at first available cycle Not for Online sensor value
        TON_OutDoorTempSnsr(
            IN := OutDoorTempSel <=1 AND NOT(TON_OutDoorTempSnsr.Q),
            PT := 10
        );

        //Selection of outdoor temperature value
        IF(TON_OutDoorTempSnsr.Q OR FirstCycle)THEN
            IF(OutDoorTempSel = OutSideTemp#OUTSIDETEMP)THEN
                OutDoorTempSnsrFilter_PreCalc[k]                   :=  Ain_Data.Fct.OutDoorTemp;
            ELSIF(OutDoorTempSel = OutSideTemp#OUTDOORUNIT)THEN
                OutDoorTempSnsrFilter_PreCalc[k]                   :=  OU_OutsideTemp;
            END_IF;

            k := k+1;

            //Indicate if temperatures has been sampled
            IF(k >= (OutDoorTempSnsr_FiltSec/10)) THEN
                IF(NOT(OutDoorTempSnsrAvgReady))THEN
                    OutDoorTempSnsrAvgReady := TRUE;
                END_IF;
                k := 0;
            END_IF;

            //Calculate temperature average
            IF(OutDoorTempSnsrAvgReady)THEN
                OutDoorTempFilterTmp := 0;
                FOR j := 0 TO (OutDoorTempSnsr_FiltSec/10) DO
                    OutDoorTempFilterTmp := OutDoorTempFilterTmp + OutDoorTempSnsrFilter_PreCalc[j];
                END_FOR;
                    OutDoorTemp := OutDoorTempFilterTmp / TO_REAL((OutDoorTempSnsr_FiltSec/10));
                    OutDoorTempFilterTmp := 0;
            ELSE
                //Calculate only sampled temperatures if not all required samples are collected
                FOR j := 0 TO (k-1) DO
                    OutDoorTempFilterTmp := OutDoorTempFilterTmp + OutDoorTempSnsrFilter_PreCalc[j];
                END_FOR;
                    OutDoorTemp := OutDoorTempFilterTmp / TO_REAL(j);
                    OutDoorTempFilterTmp := 0;
            END_IF;

            ELSIF(OutDoorTempSel = OutSideTemp#CONNECTIVITYCARD)THEN
                OutDoorTemp                     :=  Conn_OutDoorTemp;

        END_IF;

        //Update temperature value every hour or at first available cycle
        TON_OutDoorTemp(
            IN := NOT(TON_OutDoorTemp.Q),
            PT := 3600
        );

        //Selection of outdoor temperature value
        IF(TON_OutDoorTemp.Q OR FirstCycle)THEN
            OutDoorTempFilter_PreCalc[i]    :=  OutDoorTemp;

            i := i+1;

            //Indicate if temperatures has been sampled for OutDoorTemp_FiltHrs
            IF(i >= OutDoorTemp_FiltHrs) THEN
                IF(NOT(OutDoorTempAvgReady))THEN
                    OutDoorTempAvgReady := TRUE;
                END_IF;
                i := 0;
            END_IF;

            //Calculate temperature average
            IF(OutDoorTempAvgReady)THEN
                OutDoorTempFilterTmp := 0;
                FOR j := 0 TO OutDoorTemp_FiltHrs DO
                    OutDoorTempFilterTmp := OutDoorTempFilterTmp + OutDoorTempFilter_PreCalc[j];
                END_FOR;
                    OutDoorTempFilter := OutDoorTempFilterTmp / TO_REAL(OutDoorTemp_FiltHrs);
                    OutDoorTempFilterTmp := 0;
            ELSE
                //Calculate only sampled temperatures if not all required samples are collected
                FOR j := 0 TO (i-1) DO
                    OutDoorTempFilterTmp := OutDoorTempFilterTmp + OutDoorTempFilter_PreCalc[j];
                END_FOR;
                    OutDoorTempFilter := OutDoorTempFilterTmp / TO_REAL(j);
                    OutDoorTempFilterTmp := 0;
            END_IF;

        END_IF;

        IF(FirstCycle)THEN
            FirstCycle := FALSE;
        END_IF;

    {ENDREGION}

    {REGION DHW TIMING MANAGEMENT}

        /*
        If DHW regulation is required at the same time as cooling/heating, the actual regulation mode will alternate
        with a set time.
        */
        Dis_OpStateSwitch := (DHWNeed AND (OpModeAllowHeat OR OpModeAllowCool));

        TON_DHWTimer(
            IN := Dis_OpStateSwitch AND DHWFrcSwitchDone,
            PT := DhwTimerStop*60
        );
        DHWFrcSwitch := TON_DHWTimer.Q;
        DHWFrcSwitchDone  := FALSE;

        IF(DHWFrcSwitch)THEN //Select which mode that the application will transition to
            IF(HeatReq OR CoolReq) THEN     //transition to DHW
                GoToState := OpStage_Status#DHW;
            ELSE
                IF(DHWReq)THEN
                    IF(OpModeAllowHeat)THEN     //transition to heating
                        GoToState := OpStage_Status#HEATING;
                    ELSE                        //transition to cooling
                        GoToState := OpStage_Status#COOLING;
                    END_IF;
                END_IF;
            END_IF;
        END_IF;
        DHWFrcSwitchDone := (OpState = GoToState);
    {ENDREGION}

    {REGION ECT CALCULATION}
    //Select correct ECT depending on which operation mode is active, default to DHW value
        IF(GoToState = OpStage_Status#DHW)THEN
            ECT := Ain_Data.Fct.DHWBottomTemp + ECT_DHW_Offset;
        ELSIF(GoToState = OpStage_Status#HEATING)THEN
            ECT := OU_Unit.CondInTemp + ECT_Heat_Offset;
        ELSIF(GoToState = OpStage_Status#COOLING)THEN
            ECT := OU_Unit.OutDoorTemp + ECT_Cool_Offset;
        ELSE
            ECT := Ain_Data.Fct.DHWBottomTemp + ECT_DHW_Offset;
        END_IF;
        OU_Unit.ECT := ECT;
    {ENDREGION}

    {REGION DEFROST}
    IF OU_Unit.DefrostRun THEN
        GoToState := OpStage_Status#DEFROST;
    END_IF;
    {ENDREGION}

    {REGION Minimum running time}
    TON_MinRunTime(
        IN := (OpState = OpStage_Status#HEATING) OR (OpState = OpStage_Status#COOLING),
        PT := CompRunTimerMin * 60
    );
    RS_ChangeOfMode(
        S  := (OpState = OpStage_Status#HEATING) OR (OpState = OpStage_Status#COOLING),
        R1 := TON_MinRunTime.Q
    );

    MinRunTime := RS_ChangeOfMode.S AND RS_ChangeOfMode.Q1;
    {ENDREGION}

    {REGION STATE TRANSITION CHECK}
    //Only allow transition between active states if compressor temperature above ECT and if mimimum compressor time is reached
    IF(OpState <> 0 AND GoToState = 0) THEN
        OpState := 0;
    ELSE
        //Only require compressor temperature when the compressor is running
        IF(OU_CompOn)THEN
            IF (GoToState = OpStage_Status#DEFROST) THEN
                OpState := GoToState;
                OU_CompHeat := FALSE;
                SwToCoolReq := FALSE;
            ELSIF(GoToState <> OpState AND OU_CompTemp < ECT) THEN
                OU_CompHeat := TRUE;
                SwToCoolReq := FALSE;
            ELSIF(GoToState <> OpState AND MinRunTime) THEN
                OU_CompHeat := FALSE;
                SwToCoolReq := FALSE;
//            ELSIF GoToState <> OpState AND GoToState = 2 AND OU_RevValve THEN // Wants to go to cooling but needs to ramp down compressor before switch RevValve
//                SwToCoolReq := TRUE;
//            ELSIF GoToState <> OpState AND (GoToState = 1 OR GoToState = 3) AND NOT OU_RevValve THEN // Wants to go to heating or dhw but needs to ramp down compressor before switch RevValve
//                SwToCoolReq := TRUE;
            ELSIF(GoToState <> OpState) THEN
                OpState := GoToState;
                OU_CompHeat := FALSE;
                SwToCoolReq := FALSE;
            ELSE
                OU_CompHeat := FALSE;
                SwToCoolReq := FALSE;
            END_IF;

        ELSE
            OpState := GoToState;
        END_IF;
    END_IF;
    {ENDREGION}

    {REGION AUTO MODE}
    Dis_AutoMode := ManMode_Cool OR ManMode_Heat;// OR ImmHeatOnly;

    IF(UnitOn)THEN
        IF(En_AutoMode  AND NOT(Dis_AutoMode)) OR DHWFrcSwitch THEN           //AND NOT(Dis_OpStateSwitch)
            CASE OpState OF
                /*
                Change operation state depending on system need
                 0: Decision phase
                 1: Heating
                 2: Cooling
                 3: DHW
                 4: Defrost

                */

                0: //Decision phase
                    IF(DHWNeed)THEN
                        GoToState := OpStage_Status#DHW;
                    ELSIF(OpModeAllowHeat) THEN
                        GoToState := OpStage_Status#HEATING;
                    ELSIF(OpModeAllowCool)THEN
                        GoToState := OpStage_Status#COOLING;
                    END_IF;
                    //If no transition to another state is required, stop regulation
                    IF(GoToState = OpStage_Status#DECISION_PHASE)THEN
                        HeatReq := FALSE;
                        CoolReq := FALSE;
                        ImmHeatReq := FALSE;
                        DHWReq := FALSE;
                    END_IF;

                1: //Heating state
                    HeatReq := TRUE;
                    CoolReq := FALSE;
                    ImmHeatReq := FALSE;
                    DHWReq := FALSE;

                    IF OU_Unit.DefrostRun THEN
                        GoToState := OpStage_Status#DEFROST;
                    ELSIF(NOT(OpModeAllowHeat)) THEN // Return to decision phase
                        GoToState := OpStage_Status#DECISION_PHASE;
                    ELSIF(DHWNeed AND NOT DHWFrcSwitch) THEN
                        GoToState := OpStage_Status#DHW;
                    END_IF;

                2: //Cooling state
                    HeatReq := FALSE;
                    CoolReq := TRUE;
                    ImmHeatReq := FALSE;
                    DHWReq := FALSE;

                    IF(NOT(OpModeAllowCool)) THEN // Return to decision phase
                        GoToState := OpStage_Status#DECISION_PHASE;
                    ELSIF(DHWNeed) THEN
                        GoToState := OpStage_Status#DHW;
                    END_IF;
                3: //DHW
                    HeatReq := FALSE;
                    CoolReq := FALSE;
                    ImmHeatReq := FALSE;
                    DHWReq := TRUE;
                    IF OU_Unit.DefrostRun THEN
                        GoToState := OpStage_Status#DEFROST;

                    ELSIF(NOT(DHWNeed))THEN // IF statements reflects priority of the modes
                        IF OpModeAllowHeat THEN
                            GoToState := OpStage_Status#HEATING;
                        ELSIF OpModeAllowCool THEN
                            GoToState := OpStage_Status#COOLING;
                        ELSE
                            GoToState := OpStage_Status#DECISION_PHASE;
                        END_IF;
                    END_IF;
                4: //Defrost
                    HeatReq := FALSE;
                    CoolReq := FALSE;
                    ImmHeatReq := FALSE;
                    DHWReq := FALSE;
                    IF NOT OU_Unit.DefrostRun THEN  // Leave defrost mode
                        GoToState := OpStage_Status#DECISION_PHASE;
                    END_IF;

            END_CASE;
        ELSIF(Dis_AutoMode)THEN
            //Manual regulation mode
            HeatReq := ManMode_Heat;
            CoolReq := ManMode_Cool;
            ImmHeatReq := FALSE;
        ELSE //Unit off or auto mode is disabled
            HeatReq := FALSE;
            CoolReq := FALSE;
            ImmHeatReq := FALSE;
            DHWReq := FALSE;
        END_IF;
    ELSE
        HeatReq := FALSE;
        CoolReq := FALSE;
        ImmHeatReq := FALSE;
        OpState := 0;
        GoToState := 0;
    END_IF;

    {ENDREGION}

    {REGION ENERGY BALANCE CALCULATION}

    //Calculate energybalance every minute while unit is running
    TON_Energybalance(
        IN := NOT(TON_Energybalance.Q),
        PT := 1
    );
    IF(UnitOFF)THEN
        EBHP := 0;
    ELSIF(OpModeAllowHeat)THEN
        IF TON_Energybalance.Q THEN                                         //AND NOT (OpState = OpStage_Status#DHW))THEN
            IF NOT (OpState = (OpStage_Status#DHW)) THEN
                EBHP := LIMIT(EBHPMin, ((EBHP - (SupplyTempCalc - Offset_EBHP - HeatReg_Temp) / 60)), EBHPMax);
            ELSIF SupplyTempCalc > FixedEBCount THEN
                IF EBHP_Init > EBHPCompStrt AND NOT OU_Unit.CompOn THEN
                    EBHP := LIMIT((EBHPCompStrt -1), ((EBHP - (SupplyTempCalc - Offset_EBHP - FixedEBCount) / 60)), EBHPMax);             //FixedEBCount during DHW
                ELSE
                    EBHP := LIMIT((EBStepImm + EBHPCompStrt + EBHPStepOut), ((EBHP - (SupplyTempCalc - Offset_EBHP - FixedEBCount) / 60)), EBHPMax);
                END_IF;
            ELSE
                EBHP := EBHP;
            END_IF;
        ELSE
            EBHP := EBHP;
        END_IF;

        Offset_EBHP := LIMIT(0, -0.01 * EBHP, 4);
        EBCH := 0;                                                              //Energy balance for cooling = 0

        {REGION HP ALLOW START/STOP OF OUTDOOR UNIT} // EBHP logic to allow heatpump start and stop
        SR_Energybalance_HP(
            S1 := EBHP <= EBHPCompStrt AND UnitOn,
            R := (EBHP >= EBHPCompStop AND OU_Unit.CondInTemp >= SupplyTempCalc + 2) OR UnitOff OR NOT OU_CompOn
        );
        {ENDREGION}

    ELSIF((OpModeAllowCool))THEN // EBCH calculation
        IF TON_Energybalance.Q THEN
            EBCH := LIMIT(EBCHMin, ((EBCH - (SupplyTempCalcCH - Offset_EBCH - CoolReg_Temp) / 60)), EBCHMax);
        END_IF;
        Offset_EBCH := LIMIT(0, 0.01 * EBCH, 2);
        EBHP := 0;

        {REGION CH ALLOW START/STOP OF OUTDOOR UNIT} // EBCH logic to allow heatpump start and stop
        SR_Energybalance_CH(
            S1 := EBCH >= EBCHCompStrt AND UnitOn,
            R := EBCH <= EBCHCompStop OR UnitOff OR NOT OU_CompOn
        );
        {ENDREGION}
    END_IF;
    {ENDREGION}

END_PROGRAM

(* ---- 055_Protection.st ---- *)
USING System;
USING System.math;
USING Libs.Hysteresis;
USING Libs.Timer;

VAR_GLOBAL
    (**MaxTankTemp within limits*)
    MaxTankTempOk : BOOL;
    (**Comp minimum running time in heat or cool mode*)
    TON_MinTimer          : TON_s;
    (**Timer to increase flow*)
    TON_ProtectTimer          : TON_s;
        (**SR latch for Outdoor Unit freeze protection*)
        SR_OU_FreezeProt : SR;

END_VAR
PROGRAM Protection
    VAR
        (**FirstCycle*)
        FirstCycle              : BOOL := 1;
        (**Hyster MaxTankTemp*)
        HysterAdv_MaxTempTank : HysterAdv;
        (**SR latch for Climate System freeze protection*)
        SR_CS_FreezeProt : SR;
    END_VAR
{REGION MaxTankTemp}
    HysterAdv_MaxTempTank(
        In:= Ain_Data.Fct.DHWMiddleTemp ,
        SetP := MaxTankTemp,
        DiffLeft := 3.0,
        DiffRight := 0.0,
        Reverse := TRUE
    );

MaxTankTempOk := HysterAdv_MaxTempTank.Out;

{ENDREGION}

{REGION FREEZE PROTECTION CLIMATE SYTEM}
    SR_CS_FreezeProt(
        S1 := Ain_Data.Fct.OutDoorTemp < 3.5 AND NOT OpModeAllowHeat AND Ain_Data.Fct.ClimSupplyTemp < TO_REAL(SupplyTempHeatMin),
        R := (CS_FreezeProtReset OR Ain_Data.Fct.OutDoorTemp > 5)
    );
    CS_FreezeProtAct := SR_CS_FreezeProt.Q1;
{ENDREGION}

{REGION FREEZE PROTECTION OUTDOOR UNIT}
    TON_MinTimer(
        IN := SR_OU_FreezeProt.Q1,
        PT := 600
    );

    TON_ProtectTimer(
        IN := NOT TON_ProtectTimer.Q,
        PT := 10
    );

    SR_OU_FreezeProt(
        S1 := (((MIN(Ain_Data.Fct.OutDoorTemp, OU_OutsideTemp)  < 5) AND (Min(OU_CondInTemp,OU_CondOutTemp) < 5) OR OU_ComError)),
        R := (MIN(Ain_Data.Fct.OutDoorTemp, OU_OutsideTemp)  > 7 AND Min(OU_CondInTemp,OU_CondOutTemp) > 20 AND TON_MinTimer.Q)
    );
    OU_FreezeProtAct := SR_OU_FreezeProt.Q1;

    IF OU_FreezeProtAct THEN
        IF FirstCycle = 1 THEN
            PumpspdFreezeProt := PumpSpdDefrost;
            FirstCycle := 0;
        ELSIF OU_WaterFlow < OU_WaterFlowLimit AND TON_ProtectTimer.Q AND PumpspdFreezeProt < 100 THEN
            PumpspdFreezeProt := PumpspdFreezeProt + 5;
        END_IF;
    ELSIF NOT OU_FreezeProtAct THEN
        FirstCycle := 1;
    END_IF;

{ENDREGION}
END_PROGRAM

(* ---- 060_DHWRegulation.st ---- *)
USING System;
USING System.Math;
USING Libs.Math;
USING Libs.PID_Incr;
USING Libs.Timer;
USING Libs.ExpFilt;

VAR_GLOBAL
    DhwPumpMin1 : REAL;
    DhwPumpMax1 : REAL;
    DHWPumpEstimate : REAL;

    (**DHW charging period timer*)
    TON_DHWChrg       : TON_s;
    (**DHW ondelay step 2 timer*)
    TON_ChangeState      : TON_s;
    (**Extra hotwater timer*)
    TOF_ExtHotWatr     : TOF_s;
    (**Extra hotwater pulse*)
    R_Edge_tmp          : system.timer.R_Edge;
    (**PreSet dhw controller*)
    R_Edge_Dhw          : system.timer.R_Edge;
    (**Charge regulation PID*)
    DHWChrgRegPID : PID_Incr;

    temp : real;

    PumpSpdDHW              : REAL;
    (**DHW charge pump state *)
    DHWPumpState              : UINT := 0;

    DhwChrgPumpSetP         : REAL;

    DhwChrgPumpPGain        : REAL := 1;
    DhwChrgPumpIGain        : UINT := 50;
    DhwChrgPumpDGain        : UINT := 0;

        (**Circulation pump 1 timer*)
        TON_CircPump1     : TON_s;

END_VAR

PROGRAM DHWRegulation
    VAR
        (**Allow DHW*)
        AllowDHW          : BOOL;
        (**DHW top fill procent*)
        DHWTopProc        : REAL;
        (**DHW middle fill procent*)
        DHWMiddleProc     : REAL;
        (**DHW bottom fill procent*)
        DHWBottomProc     : REAL;
        (**Set/Reset DHW need*)
        SR_DHWNeed        : RS;
//        (**Charge regulation PID*)
//        DHWChrgRegPID : PID_Incr;
        (**Temperature regulation PID*)
        DHWTempRegPID : PID_Incr;
        (**DHW block from smart grid*)
        SG_DHWBlock         : BOOL;
        (**Actual Pump start setpoint*)
        ActPmpStrtSetP    : REAL;
        (**Actual Pump stop setpoint*)
        ActPmpStopSetP    : REAL;
        (**Actual Pump start temperature*)
        ActPmpStrtTemp    : REAL;
        (**Actual Pump stop temperature*)
        ActPmpStopTemp    : REAL;
        (**Index variable*)
        i                 : INT;
//        (**Heating regulation output filter*)
//        DHWReg_Filt         : ExpFilt;
        (**Circulation pump 1 low speed timer*)
        TON_GP1_LowSpd      : TON_s;
        (**Timer to increase dhw pump to increase temperature*)
        TON_DHWPumpTimer        : TON_s;
        (**PrePosition regulator*)
        PrePosDhwChrgReg    : BOOL := FALSE;
    END_VAR

    (*All the Programs are skipped while the default valeus are being installed*)
    IF RestoreDefault THEN
        RETURN;
    END_IF;

    SG_DHWBlock := SG_Status = SGStatus#BLOCKING_MODE
                    OR NOT(SystemCfg_AllowDHW);

    {REGION Extra Hot Water}
    (*Creates pulse on rising edge of ExtHotwatrEnbl**)
    R_Edge_tmp(
        In := ExtHotWatrEnbl,
        Reset := R_Edge_tmp.Out
        );
    (*Off delay to turn of after set time**)
    TOF_ExtHotWatr(
        IN := R_Edge_tmp.Out,
        PT := ExtHotWatrTime * 60
    );
    (**Disable ExtHotWatr when timer is done*)
    IF ExtHotWatrEnbl AND NOT TOF_ExtHotWatr.Q THEN
        ExtHotWatrEnbl := FALSE;
    END_IF;

    (*The extra hotwter enabled from input signal with timer or from SmartGrid [1:1]**)
    En_ExtHotWatr := ExtHotWatrEnbl OR SG_Status = SGStatus#OVERCAPACITY_MODE;

    {ENDREGION}

    {REGION START/STOP TEMPERATURES}
    //Select DHW Start/stop temperatures
    IF(DhwMode = DHWMode#ECONOMY)THEN
        DHWStartTemp := DhwEcoStartTemp;
        DHWStopTemp := DhwEcoStopTemp;
    ELSIF(DhwMode = DHWMode#COMFORT) OR (SG_Status = SGStatus#LOW_PRICE_MODE) THEN
        DHWStartTemp := DhwComfStartTemp;
        DHWStopTemp := DhwComfStopTemp;
    ELSE
        DHWStartTemp := DhwNormStartTemp;
        DHWStopTemp := DhwNormStopTemp;
    END_IF;
    {ENDREGION}

    {REGION DHWProc calculation}
        DHWTopProc := Limit(0,((Ain_Data.Fct.DHWTopTemp - DhwRefTop) / (DhwRefTopN - DhwRefTop))*100,200);
        DHWMiddleProc := Limit(0,((Ain_Data.Fct.DHWMiddleTemp - DhwRefMiddle) / (DhwRefMiddleN - DhwRefMiddle))*100,200);
        DHWBottomProc := Limit(0,((Ain_Data.Fct.DHWBottomTemp - DhwRefBottom) / (DhwRefBottomN - DhwRefBottom))*100,200);

        IF DHWTopProc = 0 THEN
            DHWProc := 0.0;
        ELSE
            DHWProc := ((DHWTopProc + DHWMiddleProc + DHWBottomProc) / 3);
        END_IF;
    {ENDREGION}

    {REGION ENABLE CHARGE}
    (**Add logic to block DHW here*)
    AllowDHW := NOT(SG_DHWBlock) AND NOT(ImmersionHeatAllow) AND (MaxTankTempOk) AND NOT (DHWCompBlock) AND NOT DHWFrcSwitch;  //Allow DHW as long as there is no blocking from smart grid -> DHW blocked if immersion heater activated by energy balance

    //Determine need of DHW
    SR_DHWNeed(                                                                                          (**DHW START CONDITIONS*)
        S := ((Ain_Data.Fct.DHWMiddleTemp < DHWStartTemp                                                   //Low middle temp.
                    OR (Ain_Data.Fct.DHWMiddleTemp<ExtHotWatrStopTemp-ExtHotWatrDiff AND En_ExtHotWatr))   //Low middle temp.(Extra hot water)
                    AND AllowDHW AND NOT TON_CircPump1.Q)                                                  //DHW is allowed

                    OR ((TON_CircPump1.Q AND Ain_Data.Fct.DHWMiddleTemp < DHWStartTemp)                               //Pump active and low top temp.
                    AND UnitOn AND AllowDHW),
                    //OR DHWProc < DHWStrtProc                                                           (**DHW STOP CONDITIONS*)
        R1  := (Ain_Data.Fct.DHWBottomTemp >= DHWStopTemp AND NOT(En_ExtHotWatr)                           //Bottom temp. reached
                    OR (Ain_Data.Fct.DHWBottomTemp>=ExtHotWatrStopTemp AND En_ExtHotWatr)                  //Bottom temp. reached(Extra hot water)
                    OR NOT(AllowDHW) OR SG_DHWBlock                                                        //DHW blocked
                    OR UnitOff)
                    //OR DHWProc >= DHWStrtProc
    );
    DHWNeed := SR_DHWNeed.Q1;

    {REGION DHW Charge Regulation}
    IF DHWChrgMode = 0 THEN                                                                     //Auto mode enabled
        IF OpState = OpStage_Status#DHW AND OU_CompOn THEN
            TON_ChangeState(
                IN := OpState = OpStage_Status#DHW AND OU_CompOn,
                PT := 20
                );
            TON_DHWPumpTimer(
                IN := NOT TON_DHWPumpTimer.Q AND TON_ChangeState.Q,
                PT := 1
            );
            IF DHWPumpState = 0 THEN                                                             //Initiation for 60 seconds the speed down pump 1% per seconds until OU_CondOut > max(45, Ain_Data.Fct.DHWMiddleTemp)
                PumpSpdDHW := 10;
                DHWPumpstate := 1;
                DHWChrgPumpSetPoint := PumpSpdDHW;
            ELSIF DHWPumpState = 1 AND TON_DHWPumpTimer.Q THEN

                DHWChrgPumpSetPoint := PumpSpdDHW;
                PumpSpdDHW := Max(PumpSpdDHW - 1,10);

                IF  OU_CondOutTemp > max(45, Ain_Data.Fct.DHWMiddleTemp) THEN                          // Change mode
                    DHWPumpState := 2;
                    PrePosDhwChrgReg := TRUE;
                END_IF;
            ELSIF DHWPumpState = 2 THEN //AND TON_DHWPumpTimer.Q AND PumpspdDHW > 10 THEN              //Fast mode to find usable dhw -> Max of 45 or middle temperature sensor.                //PumpSpdDHW := PumpSpdDHW - 1;
                DhwChrgPumpSetP := max(45, Ain_Data.Fct.DHWMiddleTemp)-Ain_Data.Fct.DHWBottomTemp;     //Delta T between Tank temp middle and bottom -> use this sensor to get a more stable regulator the using condensor in/out
                PrePosDhwChrgReg := FALSE;
                IF OU_CondOutTemp > max(45, Ain_Data.Fct.DHWMiddleTemp) AND Ain_Data.Fct.DHWBottomTemp > (OU_CondOutTemp - DHWChargeDeltaT) THEN
                    DHWPumpState := 3;

                END_IF;

            ELSIF DHWPumpState = 3 OR DHWPumpState = 4 THEN  //Delta T control

                IF DHWPumpState = 3 THEN
                    DhwChrgPumpSetP := DHWChargeDeltaT; //10;
                ELSE
                    DhwChrgPumpSetP := DHWChargeMaxEnergy; //5;
                END_IF;

                IF OU_CondOutTemp + 2 > DHWStopTemp AND OU_CondInTemp > (OU_CondOutTemp - DHWChargeDeltaT) THEN                                         //Change mood to maximize energy in tank
                    DHWPumpState := 4;
                END_IF;
            END_IF;

        ELSE
            DHWPumpState := 0;
        END_IF;
        DHWChrgRegPID(
            RegVar_PID_Incr       := OU_CondOutTemp - OU_CondInTemp,  //replaced OU_CondInTem
            SetP_PID_Incr         := DhwChrgPumpSetP,
            DeadBand_PID_Incr     := 0.0,
            Kp_PID_Incr           := TO_REAL(DhwChrgPumpPGain),
            Ti_PID_Incr           := TO_UINT(DhwChrgPumpIGain),
            Td_PID_Incr           := TO_UINT(DhwChrgPumpDGain),
            LowLim_PID_Incr       := TO_REAL(10),//DhwPumpMin1,//
            HighLim_PID_Incr      := TO_REAL(100),//DhwPumpMax1,//
            Period_PID_Incr       := 100,
            CoolHeatMode_PID_Incr := ENUM_COOL_HEAT#Cool,
            RevMode_PID_Incr      := ENUM_REV_MODE#Direct,
            ManModeVal_PID_Incr   := 0,
            En_PrePos_PID_Incr    := PrePosDhwChrgReg,
            En_ManMode_PID_Incr   := 0,
            En_PID_Incr           := TO_BOOL(DHWPumpState = 2 OR DHWPumpState = 3 OR DHWPumpState = 4)
        );

        IF DHWPumpState = 2 OR DHWPumpState = 3 OR DHWPumpState = 4 THEN
            DHWChrgPumpSetPoint := DHWChrgRegPID.Req_PID_Incr;
        END_IF;
    ELSE
        DHWChrgPumpSetPoint := PumpSpdDhwFix;                                                   //Fixed speed mode
    END_IF;

    {ENDREGION}

    //Calculation of waterflow

    //Circulation pump enable from flow
    TON_CircPump1(
        IN := WaterFlow_DHW > 1.5 AND Uniton,
        PT := TO_UINT(DhwFlowSwitchOnDel)
    );

    {ENDREGION}

    {REGION CHARGE MANAGEMENT}

        //Boost compressor towards end of DHW charge
        IF En_ExtHotWatr THEN
            DHWBoost := (To_Real(TON_DHWTimer.ET) > To_Real(DhwTimerStop) * 60 * DhwBoostPercExtHotWatr * 0.01);
        ELSE
            DHWBoost := (TO_REAL(TON_DHWTimer.ET) > To_REAL(DhwTimerStop) * 60 * DhwBoostPerc * 0.01);
        END_IF;
    {ENDREGION}

    {REGION DHW PUMP REGULATION}

    //Parameter selection for setpoint calculation
    IF(DhwMode = DHWMode#ECONOMY)THEN
        ActPmpStrtSetP := DhwSetPointStrtEco;
        ActPmpStopSetP := DhwSetPointStpEco;
        ActPmpStrtTemp := DhwBT3StrtEco;
        ActPmpStopTemp := DhwBT3StopEco;
    ELSIF(DhwMode = DHWMode#COMFORT) THEN
        ActPmpStrtSetP := DhwSetPointStrtCom;
        ActPmpStopSetP := DhwSetPointStpCom;
        ActPmpStrtTemp := DhwBT3StrtCom;
        ActPmpStopTemp := DhwBT3StopCom;
    ELSE
        ActPmpStrtSetP := DhwSetPointStrtNor;
        ActPmpStopSetP := DhwSetPointStpNor;
        ActPmpStrtTemp := DhwBT3StrtNor;
        ActPmpStopTemp := DhwBT3StopNor;
    END_IF;

    //Calculate pump regulation setpoint
    DhwPumpSetP := ScalerLimited(Ain_Data.Fct.DHWTopTemp, ActPmpStrtTemp, ActPmpStopTemp, ActPmpStrtSetP, ActPmpStopSetP);
    IF  Ain_Data.Fct.DHWTopTemp - DhwPumpSetP <= 7.5 THEN
        DHWPumpEstimate := Limit(0,(7.69 * ((WaterFlow_DHW * 1.257) - 0.85) -84.5) ,100);                         //low Delta T formula BF2 vs GP2 flow y = 1.257 x - 0.85
    ELSIF Ain_Data.Fct.DHWTopTemp - DhwPumpSetP > 7.5 AND Ain_Data.Fct.DHWTopTemp - DhwPumpSetP <=15 THEN
        DHWPumpEstimate := Limit(0,(7.69 * ((WaterFlow_DHW * 0.8621) - 0.2994)- 84.5) ,100);                      //Medium Delta T formula BF2 vs GP2 flow y = 0.8621 x - 0.2994
    ELSE
        DHWPumpEstimate := Limit(0,(7.69 * ((WaterFlow_DHW * 0.696) - 0.1418) - 84.5 ),100);                      //High Delta T formula BF2 vs GP2 flow y = 0.696 x - 0.1418
    END_IF;

    //DHWPumpEstimate :=0;
    DhwPumpMin1 := Limit(0, DHWPumpEstimate - 40, 100);   //Calculated pumpflow vs pump pwm 0-100% y= 7.69 x -84.5
    DhwPumpMax1 := Limit(0, DHWPumpEstimate + 10, 100);

    (*Preset regulator*)
    R_Edge_Dhw(
    In := TON_CircPump1.Q,
    Reset := R_Edge_Dhw.Out
    );

    (*Temperature regulation PID*)
    DHWTempRegPID(
        RegVar_PID_Incr       := Ain_Data.Fct.DHWSupplyTemp,
        SetP_PID_Incr         := DhwPumpSetP,
        DeadBand_PID_Incr     := 0.0,
        Kp_PID_Incr           := TO_REAL(DhwPumpPGain),
        Ti_PID_Incr           := TO_UINT(DhwPumpIGain),
        Td_PID_Incr           := TO_UINT(DhwPumpDGain),
        LowLim_PID_Incr       := TO_REAL(DhwPumpMin),//DhwPumpMin1,//
        HighLim_PID_Incr      := TO_REAL(DhwPumpMax),//DhwPumpMax1,//
        Period_PID_Incr       := 100,
        CoolHeatMode_PID_Incr := ENUM_COOL_HEAT#Heat,
        RevMode_PID_Incr      := ENUM_REV_MODE#Direct,
        ManModeVal_PID_Incr   := TO_REAL(PumpSpdGP2Man),
        En_PrePos_PID_Incr    := R_Edge_Dhw.Out,
        En_ManMode_PID_Incr   := PumpSpdGP2Man > 0,
        En_PID_Incr           := TON_CircPump1.Q
    );

    DHWPumpReg := DHWTempRegPID.Req_PID_Incr;

    TON_GP1_LowSpd(
        IN := TON_CircPump1.Q AND NOT(TON_GP1_LowSpd.Q),
        PT := 1
        );

    IF UnitOff OR NOT TON_CircPump1.Q  THEN // OLD: OR (DHWTempRegPID.Req_PID_Incr = 0)
        //Unit off or PID reg 0 then pump shall be set to off
        DhwCircPumpReq :=97;
    ELSIF (DHWTempRegPID.Req_PID_Incr = 0) AND TON_CircPump1.Q THEN
        IF TON_GP1_LowSpd.Q THEN
            DhwCircPumpReq := 85;
        ELSE
            DhwCircPumpReq := 97;
        END_IF;
    ELSE
        //Pump regulation
        DhwCircPumpReq := Scaler(DHWTempRegPID.Req_PID_Incr, 0, 100, 84, 10); //0-100 input is reversed and pump PWM input is scaled to fit the correct PWM curve.
    END_IF;

    Circ2Act_Req := DhwCircPumpReq;

    {ENDREGION}

END_PROGRAM

(* ---- 070_HeatingRegulation.st ---- *)
USING System;
USING System.Math;
USING Libs.Math;
USING Libs.PID_Incr;
//USING Libs.PID_ADV;
USING Libs.Timer;
USING Libs.ExpFilt;

PROGRAM HeatingRegulation
    VAR
        (**SR mode selector*)
        SR_AutoMode_Heating  : SR;
        (**Heating PID regulator*)
        PID_HeatReg          : PID_Incr;
//        (**Heating PID regulator*)
//        PID_HeatReg          : PID_Adv;
        (**Setpoint total offset*)
        SetP_Offset          : REAL;
        (**Heating blocked from smart grid*)
        SG_HeatBlock         : BOOL;
        (**Heating regulation output filter*)
        HeatReg_Filt         : ExpFilt;
        (**First Cycle done*)
        FirstCycle           : BOOL := TRUE;
        (**Shunt valve block timer*)
        TON_ShuntBlock       : TON_s;
        (**Shunt valve block pulse timer*)
        TON_ShuntBlockPulse  : TON_s;
        (**Shunt valve regulation timer*)
        TON_ShuntTimerDone   : TON_s;
        (**Shunt valve regulation factor timer*)
        TOF_ShuntFactor      : TOF_s;
        (**Shunt factor PT*)
        ShuntVlvFactor_PT    : UINT;
        (**SR shunt close*)
        SR_ShuntClose        : SR;
        (**SR shunt open*)
        SR_ShuntOpen        : SR;
        (**PID Heat Manual Value*)
        ManModeVal : REAL;
        (**Freeze time after DHW charge timer*)
        TOF_RPSBlock       : TOF_s;
        (**Setpoint calculation for Shunt control*)
        ShuntTempCalc       : REAL;
    END_VAR

    IF RestoreDefault THEN
        RETURN;
    END_IF;

    //Skip first cycle in order to avoid operating mode conflict
    IF(FirstCycle AND UnitOn)THEN
        FirstCycle := FALSE;
        RETURN;
    ELSIF(UnitOff)THEN
        FirstCycle := TRUE;
    END_IF;

    {REGION AUTOMODE}
        //Block heating/immersion heating from smart grid
        SG_HeatBlock := NOT(SystemCfg_AllowHeat);

        IF(En_AutoMode AND UnitOn)THEN
            SR_AutoMode_Heating(
                    s1 := OutDoorTempFilter < HeatModeTemp - HeatModeTempHyst
                    AND NOT(SG_HeatBlock) AND UnitON AND NOT(HeatingBlock),
                    R := OutDoorTempFilter > HeatModeTemp OR SG_HeatBlock OR UnitOff
                    );
            OpModeAllowHeat := SR_AutoMode_Heating.Q1 OR CS_FreezeProtAct;
            CS_FreezeProtReset := SR_AutoMode_Heating.Q1;
        ELSE
            OpModeAllowHeat := FALSE;
        END_IF;

    {ENDREGION}

    {REGION SETPOINT CALCULATION}

        //Add setpoint offset depending on smartgrid status
        IF(SG_Status = SGStatus#LOW_PRICE_MODE)THEN
            SG_Offset := TempSG1;
        ELSIF(SG_Status = SGStatus#OVERCAPACITY_MODE)THEN
            SG_Offset := TempSG2;
        ELSIF (SG_Status = SGStatus#BLOCKING_MODE)THEN
            SG_Offset := TempSG3;
        ELSE
            SG_Offset := 0;
        END_IF;

        //Determine total setpoint offset
        SetP_Offset := SetP_ExtAdj + SG_Offset + Offset_EBHP + HeatCurve_Offset;

        //Calculate current supply temperature setpoint
        SupplyTempCalc := LIMIT(TO_REAL(SupplyTempHeatMin), ((HeatCurve_K[Sel_HeatCurve_SetP]*OutDoorTemp) + HeatCurve_M[Sel_HeatCurve_SetP]) + SetP_Offset, TO_REAL(SupplyTempHeatMax));

    {ENDREGION}

    {REGION OU HEATING PID REGULATOR}
    //Timer to go back and freeze regulator/compressor rps after DHW charge -> test the timer and adjust
    TOF_RPSBlock(
                IN := OpState = OpStage_Status#DHW OR OpState = OpStage_Status#DEFROST,
                PT := 120
            );

    HeatReg_Temp := Ain_Data.Fct.ClimSupplyTemp;
    IF OU_CompOn THEN
        IF OU_HP_Status = 2 OR OU_HP_Status = 8 OR DHW_InitRPS = 0 THEN
            ManModeVal := ScalerLimited(OU_Unit.CurrSpd_RPS, OU_Unit.MinRPS, OU_CompMaxRps, 0.0, 100.0);
        ELSE
            ManModeVal := ScalerLimited(DHW_InitRPS, OU_Unit.MinRPS, OU_CompMaxRps, 0.0, 100.0);
        END_IF;
    ELSE
        ManModeVal := 50.0;
    END_IF;

    PID_HeatReg(
        RegVar_PID_Incr       := HeatReg_Temp,
        SetP_PID_Incr         := SupplyTempCalc,
        DeadBand_PID_Incr     := 0.0,
        Kp_PID_Incr           := TO_REAL(HeatRegPGain),
        Ti_PID_Incr           := TO_UINT(HeatRegIGain),
        Td_PID_Incr           := TO_UINT(HeatRegDGain),
        LowLim_PID_Incr       := 0.0,
        HighLim_PID_Incr      := 100.0,
        Period_PID_Incr       := 100,
        CoolHeatMode_PID_Incr := ENUM_COOL_HEAT#Heat,
        RevMode_PID_Incr      := ENUM_REV_MODE#Direct,
        ManModeVal_PID_Incr   := ManModeVal,
        En_PrePos_PID_Incr    := FALSE,
        En_ManMode_PID_Incr   := NOT OU_CompOn OR OU_HP_Status = 2 OR OU_HP_Status = 8 OR TOF_RPSBlock.Q,
        En_PID_Incr           := OpState = OpStage_Status#HEATING AND SR_Energybalance_HP.Q1
    );

    //Pass filtered request to outdoor unit
    HeatReg_Filt(
        In    := PID_HeatReg.Req_PID_Incr,
        Tau   := 50,
        En_FB := PID_HeatReg.En_PID_Incr,
        Out   => PID_HeatReq
    );

    {ENDREGION}

    {REGION SHUNT VALVE}
        //Shunt valve management
        ShuntTempCalc := Sel(ImmHeatOnly, (SupplyTempCalc - 4),SupplyTempCalc);

        IF(ShuntManMode)THEN
            ShuntVlv_Off := ShuntManClose AND NOT(ShuntManOpen);
            ShuntVlv_On := ShuntManOpen AND NOT(ShuntManClose);
        ELSIF (OpModeAllowHeat AND ((Ain_Data.Fct.DHWMiddleTemp+2) > Ain_Data.Fct.ClimSupplyTemp AND ImmersionHeatAllow AND HeatReq))
            OR (OpModeAllowHeat AND ImmHeatOnly) AND NOT(ShuntVlvBlock) THEN  //AND (((Ain_Data.Fct.DHWMiddleTemp+2) > Ain_Data.Fct.ClimSupplyTemp)

            //Invert factor calculation if supply temp is higher than setpoint
            ShuntVlvFactor_PT := SEL((ShuntTempCalc - Ain_Data.Fct.ClimSupplyTemp) < 0,
                                    TO_UINT((ShuntTempCalc - Ain_Data.Fct.ClimSupplyTemp) * ShuntVlvPFactor),
                                    TO_UINT((Ain_Data.Fct.ClimSupplyTemp - ShuntTempCalc) * ShuntVlvPFactor));

            //Calculate Shunt timer each ShuntTimeFactor minute while unit on
            TON_ShuntTimerDone(
                IN := NOT(TON_ShuntTimerDone.Q),
                PT := ShuntVlvTimeFactor
            );

            //Calculate Shunt factor -> how long steps shunt needs to take
            TOF_ShuntFactor(
                IN := TON_ShuntTimerDone.Q,
                PT := ShuntVlvFactor_PT
            );

            //Shunt closing management
            SR_ShuntClose(
                        S1 := (ShuntTempCalc < Ain_Data.Fct.ClimSupplyTemp AND TOF_ShuntFactor.Q) AND ImmersionHeatAllow,
                        R := NOT(TOF_ShuntFactor.Q) OR SR_ShuntOpen.Q1
                );
            ShuntVlv_Off := SR_ShuntClose.Q1;

            //Shunt opening management
            SR_ShuntOpen(
                        S1 := (ShuntTempCalc > Ain_Data.Fct.ClimSupplyTemp AND TOF_ShuntFactor.Q) AND ImmersionHeatAllow,
                        R := NOT(TOF_ShuntFactor.Q) OR SR_ShuntClose.Q1
                );

            ShuntVlv_On := SR_ShuntOpen.Q1;

        ELSIF(ShuntVlvBlock OR NOT ImmersionHeatAllow OR NOT OpModeAllowHeat) OR (Ain_Data.Fct.DHWMiddleTemp+2) <= Ain_Data.Fct.ClimSupplyTemp OR NOT HeatReq THEN //Block shunt valve
            ShuntVlv_On := FALSE;

            //After blocking shunt valve, force closing for X seconds
            TON_ShuntBlock(
                IN := (ShuntVlvBlock OR NOT ImmersionHeatAllow OR NOT OpModeAllowHeat) OR (Ain_Data.Fct.DHWMiddleTemp+2) <= Ain_Data.Fct.ClimSupplyTemp OR NOT HeatReq,
                PT := ShuntVlvBlock_Time
            );

            //Once inital closing procedur is complete, pulse valve closing
            IF(TON_ShuntBlock.Q)THEN
                TON_ShuntBlockPulse(
                    IN := NOT(TON_ShuntBlockPulse.Q),
                    PT := ShuntVlvBlock_PulseIntervall + ShuntVlvBlock_PulseTime
                );
            END_IF;

            ShuntVlv_Off := NOT(TON_ShuntBlock.Q)   //Initial close of valve
                            OR ((ShuntVlvBlock_PulseIntervall+ShuntVlvBlock_PulseTime) - TON_ShuntBlockPulse.ET) < ShuntVlvBlock_PulseTime; //Pulsing close command
        ELSE
            ShuntVlv_On := FALSE;
            ShuntVlv_Off := FALSE;
        END_IF;

    {ENDREGION}

END_PROGRAM

(* ---- 071_ImmersionHeater.st ---- *)
USING System;
USING System.Math;
USING Libs.Math;
USING Libs.Timer;
USING Libs.Counters;

PROGRAM ImmersionRegulation
    VAR
        (**Highest DHW start temperature*)
        ImmheatStepOutTemp   : REAL;
        (**Highest DHW stop temperature*)
        ImmheatStepInTemp    : REAL;
        (**Immersion heater step in/out timer*)
        TON_ImmHeatStep      : TON_s;
        (**Immersion heater setp in/out performed*)
        ImmheatStepDone      : BOOL := TRUE;
        (**TON imm.heater delay*)
        TOF_ImmheatEB        : TON_s;
        (** EB counter step out immersion heater*)
        SR_EB_StepOut        : SR;
        (**SR mode selector*)
        SR_AutoMode_Immheat  : SR;
        (**SR Opmode selector*)
        SR_OpMode_Immheat  : SR;
        (**Heating blocked from smart grid*)
        SG_HeatBlock         : BOOL;

    END_VAR

    SG_HeatBlock := SG_Status = SGStatus#BLOCKING_MODE
                        OR NOT(SystemCfg_AllowHeat);

    {REGION DETERMINE NEED/ALLOW}

    IF(((En_AutoMode AND UnitOn) AND NOT ImmHeatOnly)AND SystemCfg_AllowImm)AND ImmHeatStage > 0 THEN

        SR_OpMode_Immheat(
                    s1 := OutDoorTempFilter < ImmModeTemp - ImmModeTempHyst
                    AND NOT(SG_HeatBlock) AND UnitON AND NOT(HeatingBlock),
                    R := OutDoorTempFilter > ImmModeTemp OR SG_HeatBlock OR UnitOff
                    );

        OpModeAllowImm := SR_OpMode_Immheat.Q1 OR SG_Status = SGStatus#OVERCAPACITY_MODE;
    ELSIF (ImmHeatOnly) THEN
        OpModeAllowImm := TRUE;
    ELSIF (CompBlock AND CS_FreezeProtAct) THEN
        OpModeAllowImm := TRUE;
    ELSE
        OpModeAllowImm := FALSE;
    END_IF;

    {ENDREGION}

        //Immersion heater - EB counter
        //When the immersion heater has been active due to EB and EB have deactivated the immersion heater there is a high probability
        //that the immersion heater will be needed again in a short while. Because of this the system shall focus on using the outdoor unit for heating and not switching to DHW.
        TOF_ImmHeatEB(
            IN := EBHP > ((EBStepImm + EBHPCompStrt) + EBHPStepOut) AND OpmodeAllowImm,                               // Triggered when immersion heater stepsOut activated
            PT := DHWCompBlockTime*3600
            );
        SR_EB_StepOut(
                s1 := EBHP > ((EBStepImm + EBHPCompStrt) + EBHPStepOut)  AND OpmodeAllowImm AND NOT TOF_ImmHeatEB.Q,  // Triggered when immersion heater stepsOut activated
                R :=  TOF_ImmHeatEB.Q
            );
            DHWCompBlock := SR_EB_StepOut.Q1;                                                                            // Block compressor when immersion heater activated from Energy balance
        //Allow immersion heater
        SR_AutoMode_Immheat(
                s1 :=   (EBHP < (EBHPCompStrt + EBStepImm)) AND OpmodeAllowImm                                           // EB triggers immersion heater

                        OR (OU_EnvZone > 1 AND (OU_HP_Status = 2 OR OU_HP_Status = 3 OR OU_HP_Status = 4)),              // Out of ennvelope triggers immersion heater
                R := NOT SR_EB_StepOut.Q1 AND OU_EnvZone = 1 OR UnitOff OR NOT OpModeAllowImm
                );
        ImmersionHeatAllow := SR_AutoMode_Immheat.Q1 OR SG_Status = SGStatus#OVERCAPACITY_MODE OR ImmHeatOnly;

    {REGION STEP IN/OUT IMMERSION HEATER}
        //Select start/stop temperature depending if SG is in overcapacity mode or not
        ImmheatStepInTemp := SEL(SG_Status = SGStatus#OVERCAPACITY_MODE,
                            MAX(DHWStartTemp, SupplyTempCalc+3),
                            MAX(MAX(DHWStartTemp, SupplyTempCalc+3), ExtHotWatrStopTemp-ExtHotWatrDiff));

        ImmheatStepOutTemp := SEL(SG_Status = SGStatus#OVERCAPACITY_MODE,
                            MAX(DHWStopTemp, SupplyTempCalc+6),
                            MAX(MAX(DHWStopTemp, SupplyTempCalc+6), ExtHotWatrStopTemp));

        //Manual mode
        IF(ImmHeatManMode > 0 AND MaxTankTempOk)THEN
            ActImmStep := ImmHeatManMode;
        ELSIF(ImmersionHeatAllow)THEN

            //Allow in/out step with a set time intervall
            TON_ImmHeatStep(
                IN := ImmersionHeatAllow AND NOT(ImmheatStepDone),
                PT := ImmHeatStepDelay
            );

            //Reset to allow timer to start over
            IF(ImmheatStepDone)THEN
                ImmheatStepDone := FALSE;
            END_IF;

            //Only step in when we have additional steps to use
            IF(TON_ImmHeatStep.Q AND Ain_Data.Fct.DHWMiddleTemp < ImmheatStepInTemp AND ActImmStep < TO_UINT(ImmHeatStage)) THEN  // Protection against to high temperature
                ImmheatStepDone := TRUE;
                ActImmStep := ActImmStep + 1;
            //Only step out when any immersion heating steps are active
            ELSIF(TON_ImmHeatStep.Q AND Ain_Data.Fct.DHWMiddleTemp > ImmheatStepOutTemp AND ActImmStep >= 1)THEN
                ImmheatStepDone := TRUE;
                ActImmStep := ActImmStep - 1;
            END_IF;
        ELSE
            //Turn off immersion heaters
            ActImmStep := 0;

        END_IF;
    {ENDREGION}
    IF NOT MaxTankTempOk THEN
        //To high temp Turn off immersion heaters
        ActImmStep := 0;
    ELSE
        ActImmStep_Out := LIMIT(0, TO_BYTE(ActImmStep), 3);
    END_IF;

END_PROGRAM

(* ---- 080_CoolingRegulation.st ---- *)
USING System;
USING System.Math;
USING Libs.Math;
USING Libs.PID_Incr;
USING Libs.Timer;
USING Libs.ExpFilt;

PROGRAM CoolingRegulation
    VAR
        (**SR mode selector*)
        SR_AutoMode          : SR;
//        (**TON cooling delay*)
//        TON_Cooling          : TON_s;
        (**Setpoint total offset*)
        SetP_Offset          : REAL;
        (**Cooling PID regulator*)
        PID_CoolReg          : PID_Incr;
        (**Cooling regulation output filter*)
        CoolReg_Filt         : ExpFilt;
        (**PID Cool Manual Value*)
        ManModeVal : REAL;
        (**Freeze time after DHW charge timer*)
        TOF_RPSBlock       : TOF_s;
    END_VAR

    IF RestoreDefault THEN
        RETURN;
    END_IF;

//        TON_Cooling( //Cooling mode
//            IN := ((OutDoorTempFilter > CoolModeTemp) AND SystemCfg_AllowCool),
//            PT := OpModeSwitchDelay*60
//            );
        SR_AutoMode(
                s1 := ((OutDoorTempFilter > CoolModeTemp) AND SystemCfg_AllowCool),
                R := OutDoorTempFilter < CoolModeTemp - CoolModeTempHyst
                );
        OpModeAllowCool := SR_AutoMode.Q1 AND SystemCfg_AllowCool;

   //Determine total setpoint offset
        SetP_Offset := Offset_EBCH;
    //Calculate current supply temperature setpoint
        SupplyTempCalcCH := LIMIT(SupplyTempCoolMin, ((CoolCurve_K[Sel_CoolCurve_SetP]*OutDoorTemp) + CoolCurve_M[Sel_CoolCurve_SetP]) + SetP_Offset, 30);

    {REGION OU cooling PID REGULATOR}
    //Timer to go back and freeze regulator/compressor rps after DHW charge -> test the timer and adjust
    TOF_RPSBlock(
                IN := OpState = OpStage_Status#DHW OR OpState = OpStage_Status#DEFROST,
                PT := 120
            );

    CoolReg_Temp := Ain_Data.Fct.ClimSupplyTemp;
    IF OU_CompOn THEN
        IF OU_HP_Status = 2 OR OU_HP_Status = 8 OR DHW_InitRPS = 0 THEN
            ManModeVal := ScalerLimited(Max(OU_Unit.CurrSpd_RPS,50), OU_Unit.MinRPS, OU_CompMaxRps, 0.0, 100.0);
        ELSE
            ManModeVal := ScalerLimited(DHW_InitRPS, OU_Unit.MinRPS, OU_CompMaxRps, 0.0, 100.0);
        END_IF;
    ELSE
        ManModeVal := 50.0;
    END_IF;

    PID_CoolReg(
        RegVar_PID_Incr       := CoolReg_Temp,
        SetP_PID_Incr         := SupplyTempCalcCH,
        DeadBand_PID_Incr     := 0.0,
        Kp_PID_Incr           := TO_REAL(HeatRegPGain),
        Ti_PID_Incr           := TO_UINT(HeatRegIGain),
        Td_PID_Incr           := TO_UINT(HeatRegDGain),
        LowLim_PID_Incr       := 0.0,
        HighLim_PID_Incr      := 100.0,
        Period_PID_Incr       := 100,
        CoolHeatMode_PID_Incr := ENUM_COOL_HEAT#Cool,
        RevMode_PID_Incr      := ENUM_REV_MODE#Direct,
        ManModeVal_PID_Incr   := ManModeVal,
        En_PrePos_PID_Incr    := FALSE,
        En_ManMode_PID_Incr   := NOT OU_CompOn OR OU_HP_Status = 2 OR OU_HP_Status = 8 OR TOF_RPSBlock.Q,
        En_PID_Incr           := OpState = OpStage_Status#COOLING// AND SR_Energybalance.Q1
    );

    //Pass filtered request to outdoor unit
    CoolReg_Filt(
        In    := PID_CoolReg.Req_PID_Incr,
        Tau   := 50,
        En_FB := PID_CoolReg.En_PID_Incr,
        Out   => PID_CoolReq
    );
    {ENDREGION}

END_PROGRAM
